// TwinCAT 3 PLC project PLC1
// ProgramVersion: 3.1.4022.4
// libraries:
//   Tc2_EtherCAT, * (Beckhoff Automation GmbH)
//   Tc2_IoFunctions, * (Beckhoff Automation GmbH)
//   Tc2_MC2, * (Beckhoff Automation GmbH)
//   Tc2_MC2_Camming, * (Beckhoff Automation GmbH)
//   Tc2_MDP, * (Beckhoff Automation GmbH)
//   Tc2_Standard, * (Beckhoff Automation GmbH)
//   Tc2_System, * (Beckhoff Automation GmbH)
//   Tc2_TcpIp, * (Beckhoff Automation GmbH)
//   Tc2_Utilities, * (Beckhoff Automation GmbH)
//   Tc3_Module, * (Beckhoff Automation GmbH)
//   VisuDialogs, * (System)
//   VisuSymbols,3.5.10.0,System
// project tree:
//   Add-On-Instructions/ AOI_AxisAdmin.TcPOU, AOI_Bin.TcPOU, AOI_CountersAdmin.TcPOU, AOI_CylinderAdmin.TcPOU, AOI_DeltaScaraRobot.TcPOU, AOI_HeatBase.TcPOU, AOI_MS300Admin.TcPOU, AOI_SensorAdmin.TcPOU, AOI_DI.TcPOU, AOI_DO.TcPOU, AOI_Heat.TcPOU, AOI_Timer.TcPOU, AOI_VacuumAdmin.TcPOU, BLINK.TcPOU, ethercatinfo_read.TcPOU, PackMlv3_StateModel.TcPOU, SequenceTransfer.TcPOU, systeminfo_MDP_read.TcPOU
//   Data-Types/User-Defined/ Condition.TcDUT, Seq_Status.TcDUT, SocketConnect.TcDUT, UDT_BinBelt.TcDUT, UDT_BoxList.TcDUT, UDT_Hmi_AxisView.TcDUT, UDT_Hmi_OEE.TcDUT, UDT_Recipe.TcDUT, UDT_MS300Output.TcDUT, UDT_MS300Input.TcDUT, UDT_DirectMotor.TcDUT, UDT_EL3312.TcDUT, UDT_EVENT.TcDUT, UDT_AxisAdmin.TcDUT, UDT_AxisInput.TcDUT, UDT_AxisOutput.TcDUT, UDT_Box.TcDUT, UDT_CM_Condition.TcDUT, UDT_CylinderAdmin.TcDUT, UDT_CylinderInput.TcDUT, UDT_CylinderOutput.TcDUT, UDT_EM_Status.TcDUT, UDT_EM_Cmd.TcDUT, UDT_Counters.TcDUT, UDT_Hmi_Input.TcDUT, UDT_Hmi_Output.TcDUT, UDT_MS300Admin.TcDUT, UDT_MS300_REF.TcDUT, UDT_Bin.TcDUT, UDT_BinList.TcDUT, UDT_Scara.TcDUT, UDT_Scara_DI.TcDUT, UDT_Scara_DO.TcDUT, UDT_SensorAdmin.TcDUT, UDT_SensorInput.TcDUT, UDT_SensorOutput.TcDUT, UDT_UnitAdmin.TcDUT, UDT_Unit_Cmd.TcDUT, UDT_Unit_Status.TcDUT, UDT_VacuumAdmin.TcDUT, UDT_VacuumInput.TcDUT, UDT_VacuumOutput.TcDUT
//   / CommunicationTask.TcTTO, GlobalTextList.TcGTLO, IOTask.TcTTO, MotionTask.TcTTO, PlcTask1.TcTTO, 视图管理器.TcVMO (not stored)
//   POUs/Debug/ DebugPro.TcPOU
//   POUs/EtherCat/ EtherCatStates.TcPOU
//   POUs/GVLs/ ControllerTags.TcGVL
//   POUs/IO/ IO_Mapping.TcPOU
//   POUs/MG/ MotionControl.TcPOU
//   POUs/PackMaL_UN01/ EM01_Master.TcPOU, EM02_Follower1.TcPOU, EM03_Follower2.TcPOU, EM04_Follower3.TcPOU, EM05_Counters.TcPOU, EM06_Follower4_5.TcPOU, EM07_Belt6.TcPOU, EM08_Belt7.TcPOU, UN01.TcPOU
//   POUs/POUCheck/ CheckBounds.TcPOU, CheckDivDInt.TcPOU, CheckDivLInt.TcPOU, CheckDivLReal.TcPOU, CheckDivReal.TcPOU, CheckLRangeSigned.TcPOU, CheckLRangeUnsigned.TcPOU, CheckPointer.TcPOU, CheckRangeSigned.TcPOU, CheckRangeUnsigned.TcPOU
//   POUs/Socket/ Socket.TcPOU
//   VISUs/ EM.TcVIS, Vis_MAIN.TcVIS, Vis_RealAxis.TcVIS, Vis_VirtualAxis.TcVIS
//   VISUs/Part/ Visualization_Cnt.TcVIS, Vis_Axis.TcVIS, Vis_PackMlv3.TcVIS
// real-time tasks:
//   TASK PlcTask1: cycle T#10ms, priority 14, ADS port 350
//   TASK CommunicationTask: cycle T#10ms, priority 16, ADS port 351
//   TASK MotionTask: cycle T#2ms, priority 6, ADS port 352
//   TASK IOTask: cycle T#2ms, priority 8, ADS port 353
//   TASK DataTask: cycle T#50000us, priority 18, ADS port 354
//   TASK Standard: cycle T#10ms, priority 20, ADS port 355
// motion (NC):
//   TASK NC-Task 1 SAF: cycle T#2ms, priority 4, ADS port 501
//   TASK NC-Task 1 SVB: cycle T#10ms, priority 12, ADS port 511
//   AXIS V_Master (id 100)
//     General: UnitFlags=#x00000004
//     Velo: Maximum=1000
//     OtherSettings: AllowMotionCmdToSlave=true
//     encoder EncType=1
//       EncPara: ModuloFactor=200
//     drive DrvType=5
//       Analog: VeloReferenz=1000, ScaleFactorActTorque=0.1
//       TimeComp: TaskDelayCycles=1
//     controller CtrType=1
//       CtrPara: PriorControlFactor=1
//         Observer: BandWidth=20
//   AXIS Belt 4 (id 2)
//     Velo: RefSearch=35
//     OtherSettings: AllowMotionCmdToSlave=true
//     encoder EncType=19
//       EncPara: ScaleFactorNumerator=40, ScaleFactorDenominator=1280000, ModuloFactor=3300, MaxCount=#xffffffff
//     drive DrvType=16
//       DrvPara: MaxCount=#xffffffff, DriveControlDWord=#x00020100
//         Analog: ScaleFactorActTorque=0.1
//         TimeComp: TaskDelayCycles=1
//     controller CtrType=1
//       CtrPara: PriorControlFactor=1
//         Observer: BandWidth=20
//   AXIS Belt 5 (id 3)
//     Velo: RefSearch=35
//     OtherSettings: AllowMotionCmdToSlave=true
//     encoder EncType=19
//       EncPara: ScaleFactorNumerator=40, ScaleFactorDenominator=1280000, ModuloFactor=3300, MaxCount=#xffffffff
//     drive DrvType=16
//       DrvPara: MaxCount=#xffffffff, DriveControlDWord=#x00020100
//         Analog: ScaleFactorActTorque=0.1
//         TimeComp: TaskDelayCycles=1
//     controller CtrType=1
//       CtrPara: PriorControlFactor=1
//         Observer: BandWidth=20
//   AXIS Belt 6 (id 4)
//     OtherSettings: AllowMotionCmdToSlave=true
//     encoder EncType=19
//       EncPara: ScaleFactorNumerator=18.0975, ScaleFactorDenominator=1280000, Inverse=true, MaxCount=#xffffffff
//     drive DrvType=16
//       DrvPara: Inverse=true, MaxCount=#xffffffff, DriveControlDWord=#x00020100
//         Analog: ScaleFactorActTorque=0.1
//         TimeComp: TaskDelayCycles=1
//     controller CtrType=1
//       CtrPara: PriorControlFactor=1
//         Observer: BandWidth=20
//   AXIS Counter 31 (id 5)
//     General: UnitName=Degree
//     Dynamic: AccelerationMaximum=450000, DecelerationMaximum=450000
//     Velo: Maximum=20000
//     OtherSettings: AllowMotionCmdToSlave=true
//     encoder EncType=19
//       EncPara: ScaleFactorNumerator=360, ScaleFactorDenominator=1280000, MaxCount=#xffffffff
//     drive DrvType=16
//       DrvPara: MaxCount=#xffffffff, DriveControlDWord=#x00020100
//         Analog: VeloReferenz=22000, ScaleFactorActTorque=0.1
//         TimeComp: TaskDelayCycles=1
//     controller CtrType=1
//       CtrPara: PriorControlFactor=1
//         Observer: BandWidth=20
//   AXIS Counter 32 (id 6)
//     Dynamic: AccelerationMaximum=450000, DecelerationMaximum=450000
//     Velo: Maximum=20000
//     OtherSettings: AllowMotionCmdToSlave=true
//     encoder EncType=19
//       EncPara: ScaleFactorNumerator=360, ScaleFactorDenominator=1280000, MaxCount=#xffffffff
//     drive DrvType=16
//       DrvPara: MaxCount=#xffffffff, DriveControlDWord=#x00020100
//         Analog: VeloReferenz=22000, ScaleFactorActTorque=0.1
//         TimeComp: TaskDelayCycles=1
//     controller CtrType=1
//       CtrPara: PriorControlFactor=1
//         Observer: BandWidth=20
//   AXIS Counter 33 (id 7)
//     Dynamic: AccelerationMaximum=450000, DecelerationMaximum=450000
//     Velo: Maximum=20000
//     OtherSettings: AllowMotionCmdToSlave=true
//     encoder EncType=19
//       EncPara: ScaleFactorNumerator=360, ScaleFactorDenominator=1280000, MaxCount=#xffffffff
//     drive DrvType=16
//       DrvPara: MaxCount=#xffffffff, DriveControlDWord=#x00020100
//         Analog: VeloReferenz=22000, ScaleFactorActTorque=0.1
//         TimeComp: TaskDelayCycles=1
//     controller CtrType=1
//       CtrPara: PriorControlFactor=1
//         Observer: BandWidth=20
//   AXIS Counter 34 (id 8)
//     Dynamic: AccelerationMaximum=450000, DecelerationMaximum=450000
//     Velo: Maximum=20000
//     OtherSettings: AllowMotionCmdToSlave=true
//     encoder EncType=19
//       EncPara: ScaleFactorNumerator=360, ScaleFactorDenominator=1280000, MaxCount=#xffffffff
//     drive DrvType=16
//       DrvPara: MaxCount=#xffffffff, DriveControlDWord=#x00020100
//         Analog: VeloReferenz=22000, ScaleFactorActTorque=0.1
//         TimeComp: TaskDelayCycles=1
//     controller CtrType=1
//       CtrPara: PriorControlFactor=1
//         Observer: BandWidth=20
//   AXIS Counter 35 (id 9)
//     Dynamic: AccelerationMaximum=450000, DecelerationMaximum=450000
//     Velo: Maximum=20000
//     OtherSettings: AllowMotionCmdToSlave=true
//     encoder EncType=19
//       EncPara: ScaleFactorNumerator=360, ScaleFactorDenominator=1280000, MaxCount=#xffffffff
//     drive DrvType=16
//       DrvPara: MaxCount=#xffffffff, DriveControlDWord=#x00020100
//         Analog: VeloReferenz=22000, ScaleFactorActTorque=0.1
//         TimeComp: TaskDelayCycles=1
//     controller CtrType=1
//       CtrPara: PriorControlFactor=1
//         Observer: BandWidth=20
//   AXIS Counter 36 (id 10)
//     Dynamic: AccelerationMaximum=450000, DecelerationMaximum=450000
//     Velo: Maximum=20000
//     OtherSettings: AllowMotionCmdToSlave=true
//     encoder EncType=19
//       EncPara: ScaleFactorNumerator=360, ScaleFactorDenominator=1280000, MaxCount=#xffffffff
//     drive DrvType=16
//       DrvPara: MaxCount=#xffffffff, DriveControlDWord=#x00020100
//         Analog: VeloReferenz=22000, ScaleFactorActTorque=0.1
//         TimeComp: TaskDelayCycles=1
//     controller CtrType=1
//       CtrPara: PriorControlFactor=1
//         Observer: BandWidth=20
//   AXIS Counter 37 (id 11)
//     Dynamic: AccelerationMaximum=450000, DecelerationMaximum=450000
//     Velo: Maximum=20000
//     OtherSettings: AllowMotionCmdToSlave=true
//     encoder EncType=19
//       EncPara: ScaleFactorNumerator=360, ScaleFactorDenominator=1280000, MaxCount=#xffffffff
//     drive DrvType=16
//       DrvPara: MaxCount=#xffffffff, DriveControlDWord=#x00020100
//         Analog: VeloReferenz=22000, ScaleFactorActTorque=0.1
//         TimeComp: TaskDelayCycles=1
//     controller CtrType=1
//       CtrPara: PriorControlFactor=1
//         Observer: BandWidth=20
//   AXIS Counter 38 (id 12)
//     Dynamic: AccelerationMaximum=450000, DecelerationMaximum=450000
//     Velo: Maximum=20000
//     OtherSettings: AllowMotionCmdToSlave=true
//     encoder EncType=19
//       EncPara: ScaleFactorNumerator=360, ScaleFactorDenominator=1280000, MaxCount=#xffffffff
//     drive DrvType=16
//       DrvPara: MaxCount=#xffffffff, DriveControlDWord=#x00020100
//         Analog: VeloReferenz=22000, ScaleFactorActTorque=0.1
//         TimeComp: TaskDelayCycles=1
//     controller CtrType=1
//       CtrPara: PriorControlFactor=1
//         Observer: BandWidth=20
//   AXIS Counter 39 (id 13)
//     Dynamic: AccelerationMaximum=450000, DecelerationMaximum=450000
//     Velo: Maximum=20000
//     OtherSettings: AllowMotionCmdToSlave=true
//     encoder EncType=19
//       EncPara: ScaleFactorNumerator=360, ScaleFactorDenominator=1280000, MaxCount=#xffffffff
//     drive DrvType=16
//       DrvPara: MaxCount=#xffffffff, DriveControlDWord=#x00020100
//         Analog: VeloReferenz=22000, ScaleFactorActTorque=0.1
//         TimeComp: TaskDelayCycles=1
//     controller CtrType=1
//       CtrPara: PriorControlFactor=1
//         Observer: BandWidth=20
//   AXIS Counter 40 (id 14)
//     Dynamic: AccelerationMaximum=450000, DecelerationMaximum=450000
//     Velo: Maximum=20000
//     OtherSettings: AllowMotionCmdToSlave=true
//     encoder EncType=19
//       EncPara: ScaleFactorNumerator=360, ScaleFactorDenominator=1280000, MaxCount=#xffffffff
//     drive DrvType=16
//       DrvPara: MaxCount=#xffffffff, DriveControlDWord=#x00020100
//         Analog: VeloReferenz=22000, ScaleFactorActTorque=0.1
//         TimeComp: TaskDelayCycles=1
//     controller CtrType=1
//       CtrPara: PriorControlFactor=1
//         Observer: BandWidth=20
//   AXIS Belt 3 (id 15)
//     Velo: RefSearch=40
//     OtherSettings: AllowMotionCmdToSlave=true
//     encoder EncType=19
//       EncPara: ScaleFactorNumerator=40, ScaleFactorDenominator=1280000, MaxCount=#xffffffff
//     drive DrvType=16
//       DrvPara: MaxCount=#xffffffff, DriveControlDWord=#x00020100
//         Analog: ScaleFactorActTorque=0.1
//         TimeComp: TaskDelayCycles=1
//     controller CtrType=1
//       CtrPara: PriorControlFactor=1
//         Observer: BandWidth=20
//   AXIS Counter 21 (id 16)
//     Dynamic: AccelerationMaximum=450000, DecelerationMaximum=450000
//     Velo: Maximum=20000
//     OtherSettings: AllowMotionCmdToSlave=true
//     encoder EncType=19
//       EncPara: ScaleFactorNumerator=360, ScaleFactorDenominator=1280000, MaxCount=#xffffffff
//     drive DrvType=16
//       DrvPara: MaxCount=#xffffffff, DriveControlDWord=#x00020100
//         Analog: VeloReferenz=22000, ScaleFactorActTorque=0.1
//         TimeComp: TaskDelayCycles=1
//     controller CtrType=1
//       CtrPara: PriorControlFactor=1
//         Observer: BandWidth=20
//   AXIS Counter 22 (id 17)
//     Dynamic: AccelerationMaximum=450000, DecelerationMaximum=450000
//     Velo: Maximum=20000
//     OtherSettings: AllowMotionCmdToSlave=true
//     encoder EncType=19
//       EncPara: ScaleFactorNumerator=360, ScaleFactorDenominator=1280000, MaxCount=#xffffffff
//     drive DrvType=16
//       DrvPara: MaxCount=#xffffffff, DriveControlDWord=#x00020100
//         Analog: VeloReferenz=22000, ScaleFactorActTorque=0.1
//         TimeComp: TaskDelayCycles=1
//     controller CtrType=1
//       CtrPara: PriorControlFactor=1
//         Observer: BandWidth=20
//   AXIS Counter 27 (id 22)
//     Dynamic: AccelerationMaximum=450000, DecelerationMaximum=450000
//     Velo: Maximum=20000
//     OtherSettings: AllowMotionCmdToSlave=true
//     encoder EncType=19
//       EncPara: ScaleFactorNumerator=360, ScaleFactorDenominator=1280000, MaxCount=#xffffffff
//     drive DrvType=16
//       DrvPara: MaxCount=#xffffffff, DriveControlDWord=#x00020100
//         Analog: VeloReferenz=22000, ScaleFactorActTorque=0.1
//         TimeComp: TaskDelayCycles=1
//     controller CtrType=1
//       CtrPara: PriorControlFactor=1
//         Observer: BandWidth=20
//   AXIS Counter 23 (id 18)
//     Dynamic: AccelerationMaximum=450000, DecelerationMaximum=450000
//     Velo: Maximum=20000
//     OtherSettings: AllowMotionCmdToSlave=true
//     encoder EncType=19
//       EncPara: ScaleFactorNumerator=360, ScaleFactorDenominator=1280000, MaxCount=#xffffffff
//     drive DrvType=16
//       DrvPara: MaxCount=#xffffffff, DriveControlDWord=#x00020100
//         Analog: VeloReferenz=22000, ScaleFactorActTorque=0.1
//         TimeComp: TaskDelayCycles=1
//     controller CtrType=1
//       CtrPara: PriorControlFactor=1
//         Observer: BandWidth=20
//   AXIS Counter 24 (id 19)
//     Dynamic: AccelerationMaximum=450000, DecelerationMaximum=450000
//     Velo: Maximum=20000
//     OtherSettings: AllowMotionCmdToSlave=true
//     encoder EncType=19
//       EncPara: ScaleFactorNumerator=360, ScaleFactorDenominator=1280000, MaxCount=#xffffffff
//     drive DrvType=16
//       DrvPara: MaxCount=#xffffffff, DriveControlDWord=#x00020100
//         Analog: VeloReferenz=22000, ScaleFactorActTorque=0.1
//         TimeComp: TaskDelayCycles=1
//     controller CtrType=1
//       CtrPara: PriorControlFactor=1
//         Observer: BandWidth=20
//   AXIS Counter 25 (id 20)
//     Dynamic: AccelerationMaximum=450000, DecelerationMaximum=450000
//     Velo: Maximum=20000
//     OtherSettings: AllowMotionCmdToSlave=true
//     encoder EncType=19
//       EncPara: ScaleFactorNumerator=360, ScaleFactorDenominator=1280000, MaxCount=#xffffffff
//     drive DrvType=16
//       DrvPara: MaxCount=#xffffffff, DriveControlDWord=#x00020100
//         Analog: VeloReferenz=22000, ScaleFactorActTorque=0.1
//         TimeComp: TaskDelayCycles=1
//     controller CtrType=1
//       CtrPara: PriorControlFactor=1
//         Observer: BandWidth=20
//   AXIS Counter 26 (id 21)
//     Dynamic: AccelerationMaximum=450000, DecelerationMaximum=450000
//     Velo: Maximum=20000
//     OtherSettings: AllowMotionCmdToSlave=true
//     encoder EncType=19
//       EncPara: ScaleFactorNumerator=360, ScaleFactorDenominator=1280000, MaxCount=#xffffffff
//     drive DrvType=16
//       DrvPara: MaxCount=#xffffffff, DriveControlDWord=#x00020100
//         Analog: VeloReferenz=22000, ScaleFactorActTorque=0.1
//         TimeComp: TaskDelayCycles=1
//     controller CtrType=1
//       CtrPara: PriorControlFactor=1
//         Observer: BandWidth=20
//   AXIS Counter 28 (id 23)
//     Dynamic: AccelerationMaximum=450000, DecelerationMaximum=450000
//     Velo: Maximum=20000
//     OtherSettings: AllowMotionCmdToSlave=true
//     encoder EncType=19
//       EncPara: ScaleFactorNumerator=360, ScaleFactorDenominator=1280000, MaxCount=#xffffffff
//     drive DrvType=16
//       DrvPara: MaxCount=#xffffffff, DriveControlDWord=#x00020100
//         Analog: VeloReferenz=22000, ScaleFactorActTorque=0.1
//         TimeComp: TaskDelayCycles=1
//     controller CtrType=1
//       CtrPara: PriorControlFactor=1
//         Observer: BandWidth=20
//   AXIS Counter 29 (id 24)
//     Dynamic: AccelerationMaximum=450000, DecelerationMaximum=450000
//     Velo: Maximum=20000
//     OtherSettings: AllowMotionCmdToSlave=true
//     encoder EncType=19
//       EncPara: ScaleFactorNumerator=360, ScaleFactorDenominator=1280000, MaxCount=#xffffffff
//     drive DrvType=16
//       DrvPara: MaxCount=#xffffffff, DriveControlDWord=#x00020100
//         Analog: VeloReferenz=22000, ScaleFactorActTorque=0.1
//         TimeComp: TaskDelayCycles=1
//     controller CtrType=1
//       CtrPara: PriorControlFactor=1
//         Observer: BandWidth=20
//   AXIS Counter 30 (id 25)
//     Dynamic: AccelerationMaximum=450000, DecelerationMaximum=450000
//     Velo: Maximum=20000
//     OtherSettings: AllowMotionCmdToSlave=true
//     encoder EncType=19
//       EncPara: ScaleFactorNumerator=360, ScaleFactorDenominator=1280000, MaxCount=#xffffffff
//     drive DrvType=16
//       DrvPara: MaxCount=#xffffffff, DriveControlDWord=#x00020100
//         Analog: VeloReferenz=22000, ScaleFactorActTorque=0.1
//         TimeComp: TaskDelayCycles=1
//     controller CtrType=1
//       CtrPara: PriorControlFactor=1
//         Observer: BandWidth=20
//   AXIS Belt 2 (id 26)
//     Velo: RefSearch=40
//     OtherSettings: AllowMotionCmdToSlave=true
//     encoder EncType=19
//       EncPara: ScaleFactorNumerator=40, ScaleFactorDenominator=1280000, MaxCount=#xffffffff
//     drive DrvType=16
//       DrvPara: MaxCount=#xffffffff, DriveControlDWord=#x00020100
//         Analog: ScaleFactorActTorque=0.1
//         TimeComp: TaskDelayCycles=1
//     controller CtrType=1
//       CtrPara: PriorControlFactor=1
//         Observer: BandWidth=20
//   AXIS Counter 11 (id 27)
//     Dynamic: AccelerationMaximum=450000, DecelerationMaximum=450000
//     Velo: Maximum=20000
//     OtherSettings: AllowMotionCmdToSlave=true
//     encoder EncType=19
//       EncPara: ScaleFactorNumerator=360, ScaleFactorDenominator=1280000, MaxCount=#xffffffff
//     drive DrvType=16
//       DrvPara: MaxCount=#xffffffff, DriveControlDWord=#x00020100
//         Analog: VeloReferenz=22000, ScaleFactorActTorque=0.1
//         TimeComp: TaskDelayCycles=1
//     controller CtrType=1
//       CtrPara: PriorControlFactor=1
//         Observer: BandWidth=20
//   AXIS Counter 12 (id 28)
//     Dynamic: AccelerationMaximum=450000, DecelerationMaximum=450000
//     Velo: Maximum=20000
//     OtherSettings: AllowMotionCmdToSlave=true
//     encoder EncType=19
//       EncPara: ScaleFactorNumerator=360, ScaleFactorDenominator=1280000, MaxCount=#xffffffff
//     drive DrvType=16
//       DrvPara: MaxCount=#xffffffff, DriveControlDWord=#x00020100
//         Analog: VeloReferenz=22000, ScaleFactorActTorque=0.1
//         TimeComp: TaskDelayCycles=1
//     controller CtrType=1
//       CtrPara: PriorControlFactor=1
//         Observer: BandWidth=20
//   AXIS Counter 13 (id 29)
//     Dynamic: AccelerationMaximum=450000, DecelerationMaximum=450000
//     Velo: Maximum=20000
//     OtherSettings: AllowMotionCmdToSlave=true
//     encoder EncType=19
//       EncPara: ScaleFactorNumerator=360, ScaleFactorDenominator=1280000, MaxCount=#xffffffff
//     drive DrvType=16
//       DrvPara: MaxCount=#xffffffff, DriveControlDWord=#x00020100
//         Analog: VeloReferenz=22000, ScaleFactorActTorque=0.1
//         TimeComp: TaskDelayCycles=1
//     controller CtrType=1
//       CtrPara: PriorControlFactor=1
//         Observer: BandWidth=20
//   AXIS Counter 14 (id 30)
//     Dynamic: AccelerationMaximum=450000, DecelerationMaximum=450000
//     Velo: Maximum=20000
//     OtherSettings: AllowMotionCmdToSlave=true
//     encoder EncType=19
//       EncPara: ScaleFactorNumerator=360, ScaleFactorDenominator=1280000, MaxCount=#xffffffff
//     drive DrvType=16
//       DrvPara: MaxCount=#xffffffff, DriveControlDWord=#x00020100
//         Analog: VeloReferenz=22000, ScaleFactorActTorque=0.1
//         TimeComp: TaskDelayCycles=1
//     controller CtrType=1
//       CtrPara: PriorControlFactor=1
//         Observer: BandWidth=20
//   AXIS Counter 15 (id 31)
//     Dynamic: AccelerationMaximum=450000, DecelerationMaximum=450000
//     Velo: Maximum=20000
//     OtherSettings: AllowMotionCmdToSlave=true
//     encoder EncType=19
//       EncPara: ScaleFactorNumerator=360, ScaleFactorDenominator=1280000, MaxCount=#xffffffff
//     drive DrvType=16
//       DrvPara: MaxCount=#xffffffff, DriveControlDWord=#x00020100
//         Analog: VeloReferenz=22000, ScaleFactorActTorque=0.1
//         TimeComp: TaskDelayCycles=1
//     controller CtrType=1
//       CtrPara: PriorControlFactor=1
//         Observer: BandWidth=20
//   AXIS Counter 16 (id 32)
//     Dynamic: AccelerationMaximum=450000, DecelerationMaximum=450000
//     Velo: Maximum=20000
//     OtherSettings: AllowMotionCmdToSlave=true
//     encoder EncType=19
//       EncPara: ScaleFactorNumerator=360, ScaleFactorDenominator=1280000, MaxCount=#xffffffff
//     drive DrvType=16
//       DrvPara: MaxCount=#xffffffff, DriveControlDWord=#x00020100
//         Analog: VeloReferenz=22000, ScaleFactorActTorque=0.1
//         TimeComp: TaskDelayCycles=1
//     controller CtrType=1
//       CtrPara: PriorControlFactor=1
//         Observer: BandWidth=20
//   AXIS Counter 17 (id 33)
//     Dynamic: AccelerationMaximum=450000, DecelerationMaximum=450000
//     Velo: Maximum=20000
//     OtherSettings: AllowMotionCmdToSlave=true
//     encoder EncType=19
//       EncPara: ScaleFactorNumerator=360, ScaleFactorDenominator=1280000, MaxCount=#xffffffff
//     drive DrvType=16
//       DrvPara: MaxCount=#xffffffff, DriveControlDWord=#x00020100
//         Analog: VeloReferenz=22000, ScaleFactorActTorque=0.1
//         TimeComp: TaskDelayCycles=1
//     controller CtrType=1
//       CtrPara: PriorControlFactor=1
//         Observer: BandWidth=20
//   AXIS Counter 18 (id 34)
//     Dynamic: AccelerationMaximum=450000, DecelerationMaximum=450000
//     Velo: Maximum=20000
//     OtherSettings: AllowMotionCmdToSlave=true
//     encoder EncType=19
//       EncPara: ScaleFactorNumerator=360, ScaleFactorDenominator=1280000, MaxCount=#xffffffff
//     drive DrvType=16
//       DrvPara: MaxCount=#xffffffff, DriveControlDWord=#x00020100
//         Analog: VeloReferenz=22000, ScaleFactorActTorque=0.1
//         TimeComp: TaskDelayCycles=1
//     controller CtrType=1
//       CtrPara: PriorControlFactor=1
//         Observer: BandWidth=20
//   AXIS Counter 19 (id 35)
//     Dynamic: AccelerationMaximum=450000, DecelerationMaximum=450000
//     Velo: Maximum=20000
//     OtherSettings: AllowMotionCmdToSlave=true
//     encoder EncType=19
//       EncPara: ScaleFactorNumerator=360, ScaleFactorDenominator=1280000, MaxCount=#xffffffff
//     drive DrvType=16
//       DrvPara: MaxCount=#xffffffff, DriveControlDWord=#x00020100
//         Analog: VeloReferenz=22000, ScaleFactorActTorque=0.1
//         TimeComp: TaskDelayCycles=1
//     controller CtrType=1
//       CtrPara: PriorControlFactor=1
//         Observer: BandWidth=20
//   AXIS Counter 20 (id 36)
//     Dynamic: AccelerationMaximum=450000, DecelerationMaximum=450000
//     Velo: Maximum=20000
//     OtherSettings: AllowMotionCmdToSlave=true
//     encoder EncType=19
//       EncPara: ScaleFactorNumerator=360, ScaleFactorDenominator=1280000, MaxCount=#xffffffff
//     drive DrvType=16
//       DrvPara: MaxCount=#xffffffff, DriveControlDWord=#x00020100
//         Analog: VeloReferenz=22000, ScaleFactorActTorque=0.1
//         TimeComp: TaskDelayCycles=1
//     controller CtrType=1
//       CtrPara: PriorControlFactor=1
//         Observer: BandWidth=20
//   AXIS Belt 1 (id 37)
//     Velo: RefSearch=40
//     OtherSettings: AllowMotionCmdToSlave=true
//     encoder EncType=19
//       EncPara: ScaleFactorNumerator=40, ScaleFactorDenominator=1280000, MaxCount=#xffffffff
//     drive DrvType=16
//       DrvPara: MaxCount=#xffffffff, DriveControlDWord=#x00020100
//         Analog: ScaleFactorActTorque=0.1
//         TimeComp: TaskDelayCycles=1
//     controller CtrType=1
//       CtrPara: PriorControlFactor=1
//         Observer: BandWidth=20
//   AXIS Counter 1 (id 38)
//     General: UnitName=Degree
//     Dynamic: AccelerationMaximum=450000, DecelerationMaximum=450000
//     Velo: Maximum=20000
//     OtherSettings: AllowMotionCmdToSlave=true
//     encoder EncType=19
//       EncPara: ScaleFactorNumerator=360, ScaleFactorDenominator=1280000, MaxCount=#xffffffff
//     drive DrvType=16
//       DrvPara: MaxCount=#xffffffff, DriveControlDWord=#x00020100
//         Analog: VeloReferenz=22000, ScaleFactorActTorque=0.1
//         TimeComp: TaskDelayCycles=1
//     controller CtrType=1
//       CtrPara: PriorControlFactor=1
//         Observer: BandWidth=20
//   AXIS Counter 2 (id 39)
//     General: UnitName=Degree
//     Dynamic: AccelerationMaximum=450000, DecelerationMaximum=450000
//     Velo: Maximum=20000
//     OtherSettings: AllowMotionCmdToSlave=true
//     encoder EncType=19
//       EncPara: ScaleFactorNumerator=360, ScaleFactorDenominator=1280000, MaxCount=#xffffffff
//     drive DrvType=16
//       DrvPara: MaxCount=#xffffffff, DriveControlDWord=#x00020100
//         Analog: VeloReferenz=22000, ScaleFactorActTorque=0.1
//         TimeComp: TaskDelayCycles=1
//     controller CtrType=1
//       CtrPara: PriorControlFactor=1
//         Observer: BandWidth=20
//   AXIS Counter 3 (id 40)
//     General: UnitName=Degree
//     Dynamic: AccelerationMaximum=450000, DecelerationMaximum=450000
//     Velo: Maximum=20000
//     OtherSettings: AllowMotionCmdToSlave=true
//     encoder EncType=19
//       EncPara: ScaleFactorNumerator=360, ScaleFactorDenominator=1280000, MaxCount=#xffffffff
//     drive DrvType=16
//       DrvPara: MaxCount=#xffffffff, DriveControlDWord=#x00020100
//         Analog: VeloReferenz=22000, ScaleFactorActTorque=0.1
//         TimeComp: TaskDelayCycles=1
//     controller CtrType=1
//       CtrPara: PriorControlFactor=1
//         Observer: BandWidth=20
//   AXIS Counter 4 (id 41)
//     Dynamic: AccelerationMaximum=450000, DecelerationMaximum=450000
//     Velo: Maximum=20000
//     OtherSettings: AllowMotionCmdToSlave=true
//     encoder EncType=19
//       EncPara: ScaleFactorNumerator=360, ScaleFactorDenominator=1280000, MaxCount=#xffffffff
//     drive DrvType=16
//       DrvPara: MaxCount=#xffffffff, DriveControlDWord=#x00020100
//         Analog: VeloReferenz=22000, ScaleFactorActTorque=0.1
//         TimeComp: TaskDelayCycles=1
//     controller CtrType=1
//       CtrPara: PriorControlFactor=1
//         Observer: BandWidth=20
//   AXIS Counter 5 (id 42)
//     Dynamic: AccelerationMaximum=450000, DecelerationMaximum=450000
//     Velo: Maximum=20000
//     OtherSettings: AllowMotionCmdToSlave=true
//     encoder EncType=19
//       EncPara: ScaleFactorNumerator=360, ScaleFactorDenominator=1280000, MaxCount=#xffffffff
//     drive DrvType=16
//       DrvPara: MaxCount=#xffffffff, DriveControlDWord=#x00020100
//         Analog: VeloReferenz=22000, ScaleFactorActTorque=0.1
//         TimeComp: TaskDelayCycles=1
//     controller CtrType=1
//       CtrPara: PriorControlFactor=1
//         Observer: BandWidth=20
//   AXIS Counter 6 (id 43)
//     Dynamic: AccelerationMaximum=450000, DecelerationMaximum=450000
//     Velo: Maximum=20000
//     OtherSettings: AllowMotionCmdToSlave=true
//     encoder EncType=19
//       EncPara: ScaleFactorNumerator=360, ScaleFactorDenominator=1280000, MaxCount=#xffffffff
//     drive DrvType=16
//       DrvPara: MaxCount=#xffffffff, DriveControlDWord=#x00020100
//         Analog: VeloReferenz=22000, ScaleFactorActTorque=0.1
//         TimeComp: TaskDelayCycles=1
//     controller CtrType=1
//       CtrPara: PriorControlFactor=1
//         Observer: BandWidth=20
//   AXIS Counter 7 (id 44)
//     Dynamic: AccelerationMaximum=450000, DecelerationMaximum=450000
//     Velo: Maximum=20000
//     OtherSettings: AllowMotionCmdToSlave=true
//     encoder EncType=19
//       EncPara: ScaleFactorNumerator=360, ScaleFactorDenominator=1280000, MaxCount=#xffffffff
//     drive DrvType=16
//       DrvPara: MaxCount=#xffffffff, DriveControlDWord=#x00020100
//         Analog: VeloReferenz=22000, ScaleFactorActTorque=0.1
//         TimeComp: TaskDelayCycles=1
//     controller CtrType=1
//       CtrPara: PriorControlFactor=1
//         Observer: BandWidth=20
//   AXIS Counter 8 (id 45)
//     Dynamic: AccelerationMaximum=450000, DecelerationMaximum=450000
//     Velo: Maximum=20000
//     OtherSettings: AllowMotionCmdToSlave=true
//     encoder EncType=19
//       EncPara: ScaleFactorNumerator=360, ScaleFactorDenominator=1280000, MaxCount=#xffffffff
//     drive DrvType=16
//       DrvPara: MaxCount=#xffffffff, DriveControlDWord=#x00020100
//         Analog: VeloReferenz=22000, ScaleFactorActTorque=0.1
//         TimeComp: TaskDelayCycles=1
//     controller CtrType=1
//       CtrPara: PriorControlFactor=1
//         Observer: BandWidth=20
//   AXIS Counter 9 (id 46)
//     Dynamic: AccelerationMaximum=450000, DecelerationMaximum=450000
//     Velo: Maximum=20000
//     OtherSettings: AllowMotionCmdToSlave=true
//     encoder EncType=19
//       EncPara: ScaleFactorNumerator=360, ScaleFactorDenominator=1280000, MaxCount=#xffffffff
//     drive DrvType=16
//       DrvPara: MaxCount=#xffffffff, DriveControlDWord=#x00020100
//         Analog: VeloReferenz=22000, ScaleFactorActTorque=0.1
//         TimeComp: TaskDelayCycles=1
//     controller CtrType=1
//       CtrPara: PriorControlFactor=1
//         Observer: BandWidth=20
//   AXIS Counter 10 (id 47)
//     Dynamic: AccelerationMaximum=450000, DecelerationMaximum=450000
//     Velo: Maximum=20000
//     OtherSettings: AllowMotionCmdToSlave=true
//     encoder EncType=19
//       EncPara: ScaleFactorNumerator=360, ScaleFactorDenominator=1280000, MaxCount=#xffffffff
//     drive DrvType=16
//       DrvPara: MaxCount=#xffffffff, DriveControlDWord=#x00020100
//         Analog: VeloReferenz=22000, ScaleFactorActTorque=0.1
//         TimeComp: TaskDelayCycles=1
//     controller CtrType=1
//       CtrPara: PriorControlFactor=1
//         Observer: BandWidth=20
//   AXIS eAxis1 (id 101)
//     OtherSettings: AllowMotionCmdToSlave=true
//     encoder EncType=4
//       EncPara: ScaleFactorNumerator=157, ScaleFactorDenominator=1600, MaxCount=#x0000ffff
//         Inc: RefSoftSyncMask=#x0000ffff
//     drive DrvType=5
//       Analog: ScaleFactorActTorque=0.1
//       TimeComp: TaskDelayCycles=1
//     controller CtrType=1
//       CtrPara: PriorControlFactor=1
//         Observer: BandWidth=20
//   AXIS V_Master2 (id 102)
//     OtherSettings: AllowMotionCmdToSlave=true
//     encoder EncType=1
//     drive DrvType=5
//       Analog: ScaleFactorActTorque=0.1
//       TimeComp: TaskDelayCycles=1
//     controller CtrType=1
//       CtrPara: PriorControlFactor=1
//         Observer: BandWidth=20
//   AXIS Belt7 (id 48)
//     OtherSettings: AllowMotionCmdToSlave=true
//     encoder EncType=19
//       EncPara: ScaleFactorNumerator=16, ScaleFactorDenominator=1280000, Inverse=true, MaxCount=#xffffffff
//         Inc: RefSearchInverse=true
//     drive DrvType=16
//       DrvPara: Inverse=true, MaxCount=#xffffffff, DriveControlDWord=#x00020100
//         Analog: ScaleFactorActTorque=0.1
//         TimeComp: TaskDelayCycles=1
//     controller CtrType=1
//       CtrPara: PriorControlFactor=1
//         Observer: BandWidth=20
//   AXIS Puller (id 1)
//     OtherSettings: AllowMotionCmdToSlave=true
//     encoder EncType=19
//       EncPara: ScaleFactorNumerator=15.7, ScaleFactorDenominator=1280000, Inverse=true, MaxCount=#xffffffff
//     drive DrvType=16
//       DrvPara: Inverse=true, MaxCount=#xffffffff, DriveControlDWord=#x00020100
//         Analog: ScaleFactorActTorque=0.1
//         TimeComp: TaskDelayCycles=1
//     controller CtrType=1
//       CtrPara: PriorControlFactor=1
//         Observer: BandWidth=20
// I/O:
//   DEVICE Device 1 (EtherCAT), AmsNetId 5.74.170.4.2.1
//     Term 1 (EK1200) [EK1200-5000 EtherCAT Power supply (2A E-Bus)]
//       Term 2 (EL1008) [EL1008 8Ch. Dig. Input 24V, 3ms]
//       Term 3 (EL1008) [EL1008 8Ch. Dig. Input 24V, 3ms]
//       Term 4 (EL1008) [EL1008 8Ch. Dig. Input 24V, 3ms]
//       Term 5 (EL1008) [EL1008 8Ch. Dig. Input 24V, 3ms]
//       Term 6 (EL1008) [EL1008 8Ch. Dig. Input 24V, 3ms]
//       Term 7 (EL2008) [EL2008 8Ch. Dig. Output 24V, 0.5A]
//       Term 8 (EL2008) [EL2008 8Ch. Dig. Output 24V, 0.5A]
//       Term 9 (EL2008) [EL2008 8Ch. Dig. Output 24V, 0.5A]
//       Term 10 (EL2008) [EL2008 8Ch. Dig. Output 24V, 0.5A]
//       Term 11 (EL9410) [EL9410 E-Bus Power Supplier  (Diagnostics)]
//       Term 12 (EL3312) [EL3312 2Ch. Ana. Input Thermocouple (TC)]
//       Term 13 (EL3312) [EL3312 2Ch. Ana. Input Thermocouple (TC)]
//       Term 14 (EL3312) [EL3312 2Ch. Ana. Input Thermocouple (TC)]
//       Term 15 (EL3312) [EL3312 2Ch. Ana. Input Thermocouple (TC)]
//       Term 16 (EL5101) [EL5101 1Ch. Inc. Encoder 5V]
//       Term 17 (EK1122) [EK1122 2 port EtherCAT junction]
//         Drive PA14701 (ASDA-A2-E CoE Drive) [Delta ASDA-A2-E EtherCAT(CoE) Drive Rev4]
//         Drive PA14401 (ASDA-A2-E CoE Drive) [Delta ASDA-A2-E EtherCAT(CoE) Drive Rev4]
//         Drive PA14501 (ASDA-A2-E CoE Drive) [Delta ASDA-A2-E EtherCAT(CoE) Drive Rev4]
//         Drive PA14601 (ASDA-A2-E CoE Drive) [Delta ASDA-A2-E EtherCAT(CoE) Drive]
//         WPI_1(WPI_EtherCAt_32Bits) [WPI-32Bits]
//         WPI_2(WPI_EtherCAt_32Bits) [WPI-32Bits]
//         CPX_1 VI45001 (CPX-AP-I-EC-M12) [CPX-AP-I-EC-M12]
//           modules: Module 1 (CPX-AP-I-EC-M12), Module 2 (CPX-AP-I-8DI-M8-3P), Module 3 (CPX-AP-I-8DI-M8-3P), Module 4 (CPX-AP-I-8DI-M8-3P), Module 5 (CPX-AP-I-8DI-M8-3P), Module 6 (CPX-AP-I-8DI-M8-3P), Module 7 (CPX-AP-I-8DI-M8-3P), Module 8 (CPX-AP-I-8DI-M8-3P)
//       Term 22 (EK1110) [EK1110 EtherCAT extension]
//     Drive PA14901 (ASDA-A2-E CoE Drive) [Delta ASDA-A2-E EtherCAT(CoE) Drive Rev4]
//   DEVICE Device 4 (EtherCAT), AmsNetId 5.74.170.4.5.1
//     Drive PA13301 (ASDA-A2-E CoE Drive) [Delta ASDA-A2-E EtherCAT(CoE) Drive Rev4]
//     Drive PA13401 (ASDA-A2-E CoE Drive) [Delta ASDA-A2-E EtherCAT(CoE) Drive Rev4]
//     Drive PA13501 (ASDA-A2-E CoE Drive) [Delta ASDA-A2-E EtherCAT(CoE) Drive Rev4]
//     Drive PA13601 (ASDA-A2-E CoE Drive) [Delta ASDA-A2-E EtherCAT(CoE) Drive Rev4]
//     Drive PA13701 (ASDA-A2-E CoE Drive) [Delta ASDA-A2-E EtherCAT(CoE) Drive Rev4]
//     Term CIM36901 (EK1100) [EK1100 EtherCAT Coupler (2A E-Bus)]
//       Term 29 (EL1008) [EL1008 8Ch. Dig. Input 24V, 3ms]
//       Term 30 (EL1008) [EL1008 8Ch. Dig. Input 24V, 3ms]
//       Term 31 (EL1008) [EL1008 8Ch. Dig. Input 24V, 3ms]
//       Term 32 (EL1008) [EL1008 8Ch. Dig. Input 24V, 3ms]
//       Term 33 (EL1008) [EL1008 8Ch. Dig. Input 24V, 3ms]
//       Term 34 (EL1008) [EL1008 8Ch. Dig. Input 24V, 3ms]
//       Term 35 (EL1008) [EL1008 8Ch. Dig. Input 24V, 3ms]
//       Term 36 (EL1008) [EL1008 8Ch. Dig. Input 24V, 3ms]
//       Term 37 (EL2008) [EL2008 8Ch. Dig. Output 24V, 0.5A]
//       Term 38 (EL2008) [EL2008 8Ch. Dig. Output 24V, 0.5A]
//       Term 39 (EL2008) [EL2008 8Ch. Dig. Output 24V, 0.5A]
//       Term 40 (EL2008) [EL2008 8Ch. Dig. Output 24V, 0.5A]
//       Term 41 (EL2008) [EL2008 8Ch. Dig. Output 24V, 0.5A]
//       Term 42 (EL2008) [EL2008 8Ch. Dig. Output 24V, 0.5A]
//       Term 43 (EL2008) [EL2008 8Ch. Dig. Output 24V, 0.5A]
//       Term 108 (EL9011) [EL9011 End Terminal]
//     Drive PA13801 (ASDA-A2-E CoE Drive) [Delta ASDA-A2-E EtherCAT(CoE) Drive Rev4]
//     Drive PA13901 (ASDA-A2-E CoE Drive) [Delta ASDA-A2-E EtherCAT(CoE) Drive Rev4]
//     Drive PA14001 (ASDA-A2-E CoE Drive) [Delta ASDA-A2-E EtherCAT(CoE) Drive Rev4]
//     Drive PA14101 (ASDA-A2-E CoE Drive) [Delta ASDA-A2-E EtherCAT(CoE) Drive Rev4]
//     Drive PA14201 (ASDA-A2-E CoE Drive) [Delta ASDA-A2-E EtherCAT(CoE) Drive Rev4]
//     Drive PA14301 (ASDA-A2-E CoE Drive) [Delta ASDA-A2-E EtherCAT(CoE) Drive Rev4]
//     Drive PA12201 (ASDA-A2-E CoE Drive) [Delta ASDA-A2-E EtherCAT(CoE) Drive Rev4]
//     Drive PA12301 (ASDA-A2-E CoE Drive) [Delta ASDA-A2-E EtherCAT(CoE) Drive Rev4]
//     Drive PA12401 (ASDA-A2-E CoE Drive) [Delta ASDA-A2-E EtherCAT(CoE) Drive Rev4]
//     Drive PA12501 (ASDA-A2-E CoE Drive) [Delta ASDA-A2-E EtherCAT(CoE) Drive Rev4]
//     Drive PA12601 (ASDA-A2-E CoE Drive) [Delta ASDA-A2-E EtherCAT(CoE) Drive Rev4]
//     Term CIM35301 (EK1100) [EK1100 EtherCAT Coupler (2A E-Bus)]
//       Term 56 (EL1008) [EL1008 8Ch. Dig. Input 24V, 3ms]
//       Term 57 (EL1008) [EL1008 8Ch. Dig. Input 24V, 3ms]
//       Term 58 (EL1008) [EL1008 8Ch. Dig. Input 24V, 3ms]
//       Term 59 (EL1008) [EL1008 8Ch. Dig. Input 24V, 3ms]
//       Term 60 (EL1008) [EL1008 8Ch. Dig. Input 24V, 3ms]
//       Term 61 (EL1008) [EL1008 8Ch. Dig. Input 24V, 3ms]
//       Term 62 (EL1008) [EL1008 8Ch. Dig. Input 24V, 3ms]
//       Term 63 (EL1008) [EL1008 8Ch. Dig. Input 24V, 3ms]
//       Term 64 (EL2008) [EL2008 8Ch. Dig. Output 24V, 0.5A]
//       Term 65 (EL2008) [EL2008 8Ch. Dig. Output 24V, 0.5A]
//       Term 66 (EL2008) [EL2008 8Ch. Dig. Output 24V, 0.5A]
//       Term 67 (EL2008) [EL2008 8Ch. Dig. Output 24V, 0.5A]
//       Term 68 (EL2008) [EL2008 8Ch. Dig. Output 24V, 0.5A]
//       Term 69 (EL2008) [EL2008 8Ch. Dig. Output 24V, 0.5A]
//       Term 70 (EL2008) [EL2008 8Ch. Dig. Output 24V, 0.5A]
//       Term 109 (EL9011) [EL9011 End Terminal]
//     Drive PA12701 (ASDA-A2-E CoE Drive) [Delta ASDA-A2-E EtherCAT(CoE) Drive Rev4]
//     Drive PA12801 (ASDA-A2-E CoE Drive) [Delta ASDA-A2-E EtherCAT(CoE) Drive Rev4]
//     Drive PA12901 (ASDA-A2-E CoE Drive) [Delta ASDA-A2-E EtherCAT(CoE) Drive Rev4]
//     Drive PA13001 (ASDA-A2-E CoE Drive) [Delta ASDA-A2-E EtherCAT(CoE) Drive Rev4]
//     Drive PA13101 (ASDA-A2-E CoE Drive) [Delta ASDA-A2-E EtherCAT(CoE) Drive Rev4]
//     Drive PA13201 (ASDA-A2-E CoE Drive) [Delta ASDA-A2-E EtherCAT(CoE) Drive Rev4]
//     Drive PA11101 (ASDA-A2-E CoE Drive) [Delta ASDA-A2-E EtherCAT(CoE) Drive Rev4]
//     Drive PA11201 (ASDA-A2-E CoE Drive) [Delta ASDA-A2-E EtherCAT(CoE) Drive Rev4]
//     Drive PA11301 (ASDA-A2-E CoE Drive) [Delta ASDA-A2-E EtherCAT(CoE) Drive Rev4]
//     Drive PA11401 (ASDA-A2-E CoE Drive) [Delta ASDA-A2-E EtherCAT(CoE) Drive Rev4]
//     Drive PA11501 (ASDA-A2-E CoE Drive) [Delta ASDA-A2-E EtherCAT(CoE) Drive Rev4]
//     Term CIM33701 (EK1100) [EK1100 EtherCAT Coupler (2A E-Bus)]
//       Term 83 (EL1008) [EL1008 8Ch. Dig. Input 24V, 3ms]
//       Term 84 (EL1008) [EL1008 8Ch. Dig. Input 24V, 3ms]
//       Term 85 (EL1008) [EL1008 8Ch. Dig. Input 24V, 3ms]
//       Term 86 (EL1008) [EL1008 8Ch. Dig. Input 24V, 3ms]
//       Term 87 (EL1008) [EL1008 8Ch. Dig. Input 24V, 3ms]
//       Term 88 (EL1008) [EL1008 8Ch. Dig. Input 24V, 3ms]
//       Term 89 (EL1008) [EL1008 8Ch. Dig. Input 24V, 3ms]
//       Term 90 (EL1008) [EL1008 8Ch. Dig. Input 24V, 3ms]
//       Term 91 (EL2008) [EL2008 8Ch. Dig. Output 24V, 0.5A]
//       Term 92 (EL2008) [EL2008 8Ch. Dig. Output 24V, 0.5A]
//       Term 93 (EL2008) [EL2008 8Ch. Dig. Output 24V, 0.5A]
//       Term 94 (EL2008) [EL2008 8Ch. Dig. Output 24V, 0.5A]
//       Term 95 (EL2008) [EL2008 8Ch. Dig. Output 24V, 0.5A]
//       Term 96 (EL2008) [EL2008 8Ch. Dig. Output 24V, 0.5A]
//       Term 97 (EL2008) [EL2008 8Ch. Dig. Output 24V, 0.5A]
//       Term 110 (EL9011) [EL9011 End Terminal]
//     Drive PA11601 (ASDA-A2-E CoE Drive) [Delta ASDA-A2-E EtherCAT(CoE) Drive Rev4]
//     Drive PA11701 (ASDA-A2-E CoE Drive) [Delta ASDA-A2-E EtherCAT(CoE) Drive Rev4]
//     Drive PA11801 (ASDA-A2-E CoE Drive) [Delta ASDA-A2-E EtherCAT(CoE) Drive Rev4]
//     Drive PA11901 (ASDA-A2-E CoE Drive) [Delta ASDA-A2-E EtherCAT(CoE) Drive Rev4]
//     Drive PA12001 (ASDA-A2-E CoE Drive) [Delta ASDA-A2-E EtherCAT(CoE) Drive Rev4]
//     Drive PA12101 (ASDA-A2-E CoE Drive) [Delta ASDA-A2-E EtherCAT(CoE) Drive Rev4]
//     Drive PA10101 (ASDA-A2-E CoE Drive) [Delta ASDA-A2-E EtherCAT(CoE) Drive Rev4]
//     Drive PA10201 (ASDA-A2-E CoE Drive) [Delta ASDA-A2-E EtherCAT(CoE) Drive Rev4]
//     Drive PA10301 (ASDA-A2-E CoE Drive) [Delta ASDA-A2-E EtherCAT(CoE) Drive Rev4]
//     Drive PA10401 (ASDA-A2-E CoE Drive) [Delta ASDA-A2-E EtherCAT(CoE) Drive Rev4]
//     Drive PA10501 (ASDA-A2-E CoE Drive) [Delta ASDA-A2-E EtherCAT(CoE) Drive Rev4]
//     Term CIM32101 (EK1100) [EK1100 EtherCAT Coupler (2A E-Bus)]
//       Term 110 (EL1008) [EL1008 8Ch. Dig. Input 24V, 3ms]
//       Term 111 (EL1008) [EL1008 8Ch. Dig. Input 24V, 3ms]
//       Term 112 (EL1008) [EL1008 8Ch. Dig. Input 24V, 3ms]
//       Term 113 (EL1008) [EL1008 8Ch. Dig. Input 24V, 3ms]
//       Term 114 (EL1008) [EL1008 8Ch. Dig. Input 24V, 3ms]
//       Term 115 (EL1008) [EL1008 8Ch. Dig. Input 24V, 3ms]
//       Term 116 (EL1008) [EL1008 8Ch. Dig. Input 24V, 3ms]
//       Term 117 (EL1008) [EL1008 8Ch. Dig. Input 24V, 3ms]
//       Term 118 (EL2008) [EL2008 8Ch. Dig. Output 24V, 0.5A]
//       Term 119 (EL2008) [EL2008 8Ch. Dig. Output 24V, 0.5A]
//       Term 120 (EL2008) [EL2008 8Ch. Dig. Output 24V, 0.5A]
//       Term 121 (EL2008) [EL2008 8Ch. Dig. Output 24V, 0.5A]
//       Term 122 (EL2008) [EL2008 8Ch. Dig. Output 24V, 0.5A]
//       Term 123 (EL2008) [EL2008 8Ch. Dig. Output 24V, 0.5A]
//       Term 124 (EL2008) [EL2008 8Ch. Dig. Output 24V, 0.5A]
//       Term 111 (EL9011) [EL9011 End Terminal]
//     Drive PA10601 (ASDA-A2-E CoE Drive) [Delta ASDA-A2-E EtherCAT(CoE) Drive Rev4]
//     Drive PA10701 (ASDA-A2-E CoE Drive) [Delta ASDA-A2-E EtherCAT(CoE) Drive Rev4]
//     Drive PA10801 (ASDA-A2-E CoE Drive) [Delta ASDA-A2-E EtherCAT(CoE) Drive Rev4]
//     Drive PA10901 (ASDA-A2-E CoE Drive) [Delta ASDA-A2-E EtherCAT(CoE) Drive Rev4]
//     Drive PA11001 (ASDA-A2-E CoE Drive) [Delta ASDA-A2-E EtherCAT(CoE) Drive Rev4]
//   DEVICE Device 6 (NOV-DP-RAM)
//     Box 18 (Retain Handler)
// variable links:
//   NC-Task 1 SAF/Axes/Belt 1 <-> Device 4 (EtherCAT)/Drive PA12101 (ASDA-A2-E CoE Drive)
//     Drive/Inputs/In/nDataIn3[0] <-> 1st TxPDO Mapping/ActualTorque
//     Drive/Inputs/In/nDcOutputTime <-> InfoData/DcOutputShift
//     Drive/Inputs/In/nState1 <-> 1st TxPDO Mapping/Status Word
//     Drive/Inputs/In/nState2 <-> 1st TxPDO Mapping/Status Word @bit 8
//     Drive/Inputs/In/nState4 @bit 1 <-> WcState/InputToggle
//     Drive/Inputs/In/nState4 <-> WcState/WcState
//     Drive/Outputs/Out/nCtrl1 <-> 2nd RxPDO Mapping/Control Word
//     Drive/Outputs/Out/nCtrl2 <-> 2nd RxPDO Mapping/Control Word @bit 8
//     Drive/Outputs/Out/nDataOut1 <-> 2nd RxPDO Mapping/TargetPosition
//     Enc/Inputs/In/nDataIn1 <-> 1st TxPDO Mapping/ActualPosition
//     Enc/Inputs/In/nDataIn7 <-> 1st TxPDO Mapping/Velocity actual value
//     Enc/Inputs/In/nDcInputTime <-> InfoData/DcInputShift
//     Enc/Inputs/In/nState4 @bit 1 <-> WcState/InputToggle
//     Enc/Inputs/In/nState4 <-> WcState/WcState
//   NC-Task 1 SAF/Axes/Belt 2 <-> Device 4 (EtherCAT)/Drive PA13201 (ASDA-A2-E CoE Drive)
//     Drive/Inputs/In/nDataIn3[0] <-> 1st TxPDO Mapping/ActualTorque
//     Drive/Inputs/In/nDcOutputTime <-> InfoData/DcOutputShift
//     Drive/Inputs/In/nState1 <-> 1st TxPDO Mapping/Status Word
//     Drive/Inputs/In/nState2 <-> 1st TxPDO Mapping/Status Word @bit 8
//     Drive/Inputs/In/nState4 @bit 1 <-> WcState/InputToggle
//     Drive/Inputs/In/nState4 <-> WcState/WcState
//     Drive/Outputs/Out/nCtrl1 <-> 2nd RxPDO Mapping/Control Word
//     Drive/Outputs/Out/nCtrl2 <-> 2nd RxPDO Mapping/Control Word @bit 8
//     Drive/Outputs/Out/nDataOut1 <-> 2nd RxPDO Mapping/TargetPosition
//     Enc/Inputs/In/nDataIn1 <-> 1st TxPDO Mapping/ActualPosition
//     Enc/Inputs/In/nDataIn7 <-> 1st TxPDO Mapping/Velocity actual value
//     Enc/Inputs/In/nDcInputTime <-> InfoData/DcInputShift
//     Enc/Inputs/In/nState4 @bit 1 <-> WcState/InputToggle
//     Enc/Inputs/In/nState4 <-> WcState/WcState
//   NC-Task 1 SAF/Axes/Belt 3 <-> Device 4 (EtherCAT)/Drive PA14301 (ASDA-A2-E CoE Drive)
//     Drive/Inputs/In/nDataIn3[0] <-> 1st TxPDO Mapping/ActualTorque
//     Drive/Inputs/In/nDcOutputTime <-> InfoData/DcOutputShift
//     Drive/Inputs/In/nState1 <-> 1st TxPDO Mapping/Status Word
//     Drive/Inputs/In/nState2 <-> 1st TxPDO Mapping/Status Word @bit 8
//     Drive/Inputs/In/nState4 @bit 1 <-> WcState/InputToggle
//     Drive/Inputs/In/nState4 <-> WcState/WcState
//     Drive/Outputs/Out/nCtrl1 <-> 2nd RxPDO Mapping/Control Word
//     Drive/Outputs/Out/nCtrl2 <-> 2nd RxPDO Mapping/Control Word @bit 8
//     Drive/Outputs/Out/nDataOut1 <-> 2nd RxPDO Mapping/TargetPosition
//     Enc/Inputs/In/nDataIn1 <-> 1st TxPDO Mapping/ActualPosition
//     Enc/Inputs/In/nDataIn7 <-> 1st TxPDO Mapping/Velocity actual value
//     Enc/Inputs/In/nDcInputTime <-> InfoData/DcInputShift
//     Enc/Inputs/In/nState4 @bit 1 <-> WcState/InputToggle
//     Enc/Inputs/In/nState4 <-> WcState/WcState
//   NC-Task 1 SAF/Axes/Belt 4 <-> Device 1 (EtherCAT)/Term 1 (EK1200)/Term 17 (EK1122)/Drive PA14401 (ASDA-A2-E CoE Drive)
//     Drive/Inputs/In/nDataIn3[0] <-> 1st Transmit PDO Mapping/Torque actual value
//     Drive/Inputs/In/nDcOutputTime <-> InfoData/DcOutputShift
//     Drive/Inputs/In/nState1 <-> 1st Transmit PDO Mapping/Statusword
//     Drive/Inputs/In/nState2 <-> 1st Transmit PDO Mapping/Statusword @bit 8
//     Drive/Inputs/In/nState4 @bit 1 <-> WcState/InputToggle
//     Drive/Inputs/In/nState4 <-> WcState/WcState
//     Drive/Outputs/Out/nCtrl1 <-> 2nd Receive PDO Mapping/Controlword
//     Drive/Outputs/Out/nCtrl2 <-> 2nd Receive PDO Mapping/Controlword @bit 8
//     Drive/Outputs/Out/nDataOut1 <-> 2nd Receive PDO Mapping/Target position
//     Enc/Inputs/In/nDataIn1 <-> 1st Transmit PDO Mapping/Position actual value
//     Enc/Inputs/In/nDataIn7 <-> 1st Transmit PDO Mapping/Velocity actual value
//     Enc/Inputs/In/nDcInputTime <-> InfoData/DcInputShift
//     Enc/Inputs/In/nState4 @bit 1 <-> WcState/InputToggle
//     Enc/Inputs/In/nState4 <-> WcState/WcState
//   NC-Task 1 SAF/Axes/Belt 5 <-> Device 1 (EtherCAT)/Term 1 (EK1200)/Term 17 (EK1122)/Drive PA14501 (ASDA-A2-E CoE Drive)
//     Drive/Inputs/In/nDataIn3[0] <-> 1st Transmit PDO Mapping/Torque actual value
//     Drive/Inputs/In/nDcOutputTime <-> InfoData/DcOutputShift
//     Drive/Inputs/In/nState1 <-> 1st Transmit PDO Mapping/Statusword
//     Drive/Inputs/In/nState2 <-> 1st Transmit PDO Mapping/Statusword @bit 8
//     Drive/Inputs/In/nState4 @bit 1 <-> WcState/InputToggle
//     Drive/Inputs/In/nState4 <-> WcState/WcState
//     Drive/Outputs/Out/nCtrl1 <-> 2nd Receive PDO Mapping/Controlword
//     Drive/Outputs/Out/nCtrl2 <-> 2nd Receive PDO Mapping/Controlword @bit 8
//     Drive/Outputs/Out/nDataOut1 <-> 2nd Receive PDO Mapping/Target position
//     Enc/Inputs/In/nDataIn1 <-> 1st Transmit PDO Mapping/Position actual value
//     Enc/Inputs/In/nDataIn7 <-> 1st Transmit PDO Mapping/Velocity actual value
//     Enc/Inputs/In/nDcInputTime <-> InfoData/DcInputShift
//     Enc/Inputs/In/nState4 @bit 1 <-> WcState/InputToggle
//     Enc/Inputs/In/nState4 <-> WcState/WcState
//   NC-Task 1 SAF/Axes/Belt 6 <-> Device 1 (EtherCAT)/Term 1 (EK1200)/Term 17 (EK1122)/Drive PA14601 (ASDA-A2-E CoE Drive)
//     Drive/Inputs/In/nDataIn3[0] <-> 1st TxPDO Mapping/ActualTorque
//     Drive/Inputs/In/nDcOutputTime <-> InfoData/DcOutputShift
//     Drive/Inputs/In/nState1 <-> 1st TxPDO Mapping/Status Word
//     Drive/Inputs/In/nState2 <-> 1st TxPDO Mapping/Status Word @bit 8
//     Drive/Inputs/In/nState4 @bit 1 <-> WcState/InputToggle
//     Drive/Inputs/In/nState4 <-> WcState/WcState
//     Drive/Outputs/Out/nCtrl1 <-> 2nd RxPDO Mapping/Control Word
//     Drive/Outputs/Out/nCtrl2 <-> 2nd RxPDO Mapping/Control Word @bit 8
//     Drive/Outputs/Out/nDataOut1 <-> 2nd RxPDO Mapping/TargetPosition
//     Enc/Inputs/In/nDataIn1 <-> 1st TxPDO Mapping/ActualPosition
//     Enc/Inputs/In/nDataIn7 <-> 1st TxPDO Mapping/Velocity actual value
//     Enc/Inputs/In/nDcInputTime <-> InfoData/DcInputShift
//     Enc/Inputs/In/nState4 @bit 1 <-> WcState/InputToggle
//     Enc/Inputs/In/nState4 <-> WcState/WcState
//   NC-Task 1 SAF/Axes/Belt7 <-> Device 1 (EtherCAT)/Drive PA14901 (ASDA-A2-E CoE Drive)
//     Drive/Inputs/In/nDataIn3[0] <-> 1st TxPDO Mapping/ActualTorque
//     Drive/Inputs/In/nDcOutputTime <-> InfoData/DcOutputShift
//     Drive/Inputs/In/nState1 <-> 1st TxPDO Mapping/Status Word
//     Drive/Inputs/In/nState2 <-> 1st TxPDO Mapping/Status Word @bit 8
//     Drive/Inputs/In/nState4 @bit 1 <-> WcState/InputToggle
//     Drive/Inputs/In/nState4 <-> WcState/WcState
//     Drive/Outputs/Out/nCtrl1 <-> 2nd RxPDO Mapping/Control Word
//     Drive/Outputs/Out/nCtrl2 <-> 2nd RxPDO Mapping/Control Word @bit 8
//     Drive/Outputs/Out/nDataOut1 <-> 2nd RxPDO Mapping/TargetPosition
//     Enc/Inputs/In/nDataIn1 <-> 1st TxPDO Mapping/ActualPosition
//     Enc/Inputs/In/nDataIn7 <-> 1st TxPDO Mapping/Velocity actual value
//     Enc/Inputs/In/nDcInputTime <-> InfoData/DcInputShift
//     Enc/Inputs/In/nState4 @bit 1 <-> WcState/InputToggle
//     Enc/Inputs/In/nState4 <-> WcState/WcState
//   NC-Task 1 SAF/Axes/Counter 1 <-> Device 4 (EtherCAT)/Drive PA10101 (ASDA-A2-E CoE Drive)
//     Drive/Inputs/In/nDataIn3[0] <-> 1st TxPDO Mapping/ActualTorque
//     Drive/Inputs/In/nDcOutputTime <-> InfoData/DcOutputShift
//     Drive/Inputs/In/nState1 <-> 1st TxPDO Mapping/Status Word
//     Drive/Inputs/In/nState2 <-> 1st TxPDO Mapping/Status Word @bit 8
//     Drive/Inputs/In/nState4 @bit 1 <-> WcState/InputToggle
//     Drive/Inputs/In/nState4 <-> WcState/WcState
//     Drive/Outputs/Out/nCtrl1 <-> 2nd RxPDO Mapping/Control Word
//     Drive/Outputs/Out/nCtrl2 <-> 2nd RxPDO Mapping/Control Word @bit 8
//     Drive/Outputs/Out/nDataOut1 <-> 2nd RxPDO Mapping/TargetPosition
//     Enc/Inputs/In/nDataIn1 <-> 1st TxPDO Mapping/ActualPosition
//     Enc/Inputs/In/nDataIn7 <-> 1st TxPDO Mapping/Velocity actual value
//     Enc/Inputs/In/nDcInputTime <-> InfoData/DcInputShift
//     Enc/Inputs/In/nState4 @bit 1 <-> WcState/InputToggle
//     Enc/Inputs/In/nState4 <-> WcState/WcState
//   NC-Task 1 SAF/Axes/Counter 10 <-> Device 4 (EtherCAT)/Drive PA11001 (ASDA-A2-E CoE Drive)
//     Drive/Inputs/In/nDataIn3[0] <-> 1st TxPDO Mapping/ActualTorque
//     Drive/Inputs/In/nDcOutputTime <-> InfoData/DcOutputShift
//     Drive/Inputs/In/nState1 <-> 1st TxPDO Mapping/Status Word
//     Drive/Inputs/In/nState2 <-> 1st TxPDO Mapping/Status Word @bit 8
//     Drive/Inputs/In/nState4 @bit 1 <-> WcState/InputToggle
//     Drive/Inputs/In/nState4 <-> WcState/WcState
//     Drive/Outputs/Out/nCtrl1 <-> 2nd RxPDO Mapping/Control Word
//     Drive/Outputs/Out/nCtrl2 <-> 2nd RxPDO Mapping/Control Word @bit 8
//     Drive/Outputs/Out/nDataOut1 <-> 2nd RxPDO Mapping/TargetPosition
//     Enc/Inputs/In/nDataIn1 <-> 1st TxPDO Mapping/ActualPosition
//     Enc/Inputs/In/nDataIn7 <-> 1st TxPDO Mapping/Velocity actual value
//     Enc/Inputs/In/nDcInputTime <-> InfoData/DcInputShift
//     Enc/Inputs/In/nState4 @bit 1 <-> WcState/InputToggle
//     Enc/Inputs/In/nState4 <-> WcState/WcState
//   NC-Task 1 SAF/Axes/Counter 11 <-> Device 4 (EtherCAT)/Drive PA11101 (ASDA-A2-E CoE Drive)
//     Drive/Inputs/In/nDataIn3[0] <-> 1st TxPDO Mapping/ActualTorque
//     Drive/Inputs/In/nDcOutputTime <-> InfoData/DcOutputShift
//     Drive/Inputs/In/nState1 <-> 1st TxPDO Mapping/Status Word
//     Drive/Inputs/In/nState2 <-> 1st TxPDO Mapping/Status Word @bit 8
//     Drive/Inputs/In/nState4 @bit 1 <-> WcState/InputToggle
//     Drive/Inputs/In/nState4 <-> WcState/WcState
//     Drive/Outputs/Out/nCtrl1 <-> 2nd RxPDO Mapping/Control Word
//     Drive/Outputs/Out/nCtrl2 <-> 2nd RxPDO Mapping/Control Word @bit 8
//     Drive/Outputs/Out/nDataOut1 <-> 2nd RxPDO Mapping/TargetPosition
//     Enc/Inputs/In/nDataIn1 <-> 1st TxPDO Mapping/ActualPosition
//     Enc/Inputs/In/nDataIn7 <-> 1st TxPDO Mapping/Velocity actual value
//     Enc/Inputs/In/nDcInputTime <-> InfoData/DcInputShift
//     Enc/Inputs/In/nState4 @bit 1 <-> WcState/InputToggle
//     Enc/Inputs/In/nState4 <-> WcState/WcState
//   NC-Task 1 SAF/Axes/Counter 12 <-> Device 4 (EtherCAT)/Drive PA11201 (ASDA-A2-E CoE Drive)
//     Drive/Inputs/In/nDataIn3[0] <-> 1st TxPDO Mapping/ActualTorque
//     Drive/Inputs/In/nDcOutputTime <-> InfoData/DcOutputShift
//     Drive/Inputs/In/nState1 <-> 1st TxPDO Mapping/Status Word
//     Drive/Inputs/In/nState2 <-> 1st TxPDO Mapping/Status Word @bit 8
//     Drive/Inputs/In/nState4 @bit 1 <-> WcState/InputToggle
//     Drive/Inputs/In/nState4 <-> WcState/WcState
//     Drive/Outputs/Out/nCtrl1 <-> 2nd RxPDO Mapping/Control Word
//     Drive/Outputs/Out/nCtrl2 <-> 2nd RxPDO Mapping/Control Word @bit 8
//     Drive/Outputs/Out/nDataOut1 <-> 2nd RxPDO Mapping/TargetPosition
//     Enc/Inputs/In/nDataIn1 <-> 1st TxPDO Mapping/ActualPosition
//     Enc/Inputs/In/nDataIn7 <-> 1st TxPDO Mapping/Velocity actual value
//     Enc/Inputs/In/nDcInputTime <-> InfoData/DcInputShift
//     Enc/Inputs/In/nState4 @bit 1 <-> WcState/InputToggle
//     Enc/Inputs/In/nState4 <-> WcState/WcState
//   NC-Task 1 SAF/Axes/Counter 13 <-> Device 4 (EtherCAT)/Drive PA11301 (ASDA-A2-E CoE Drive)
//     Drive/Inputs/In/nDataIn3[0] <-> 1st TxPDO Mapping/ActualTorque
//     Drive/Inputs/In/nDcOutputTime <-> InfoData/DcOutputShift
//     Drive/Inputs/In/nState1 <-> 1st TxPDO Mapping/Status Word
//     Drive/Inputs/In/nState2 <-> 1st TxPDO Mapping/Status Word @bit 8
//     Drive/Inputs/In/nState4 @bit 1 <-> WcState/InputToggle
//     Drive/Inputs/In/nState4 <-> WcState/WcState
//     Drive/Outputs/Out/nCtrl1 <-> 2nd RxPDO Mapping/Control Word
//     Drive/Outputs/Out/nCtrl2 <-> 2nd RxPDO Mapping/Control Word @bit 8
//     Drive/Outputs/Out/nDataOut1 <-> 2nd RxPDO Mapping/TargetPosition
//     Enc/Inputs/In/nDataIn1 <-> 1st TxPDO Mapping/ActualPosition
//     Enc/Inputs/In/nDataIn7 <-> 1st TxPDO Mapping/Velocity actual value
//     Enc/Inputs/In/nDcInputTime <-> InfoData/DcInputShift
//     Enc/Inputs/In/nState4 @bit 1 <-> WcState/InputToggle
//     Enc/Inputs/In/nState4 <-> WcState/WcState
//   NC-Task 1 SAF/Axes/Counter 14 <-> Device 4 (EtherCAT)/Drive PA11401 (ASDA-A2-E CoE Drive)
//     Drive/Inputs/In/nDataIn3[0] <-> 1st TxPDO Mapping/ActualTorque
//     Drive/Inputs/In/nDcOutputTime <-> InfoData/DcOutputShift
//     Drive/Inputs/In/nState1 <-> 1st TxPDO Mapping/Status Word
//     Drive/Inputs/In/nState2 <-> 1st TxPDO Mapping/Status Word @bit 8
//     Drive/Inputs/In/nState4 @bit 1 <-> WcState/InputToggle
//     Drive/Inputs/In/nState4 <-> WcState/WcState
//     Drive/Outputs/Out/nCtrl1 <-> 2nd RxPDO Mapping/Control Word
//     Drive/Outputs/Out/nCtrl2 <-> 2nd RxPDO Mapping/Control Word @bit 8
//     Drive/Outputs/Out/nDataOut1 <-> 2nd RxPDO Mapping/TargetPosition
//     Enc/Inputs/In/nDataIn1 <-> 1st TxPDO Mapping/ActualPosition
//     Enc/Inputs/In/nDataIn7 <-> 1st TxPDO Mapping/Velocity actual value
//     Enc/Inputs/In/nDcInputTime <-> InfoData/DcInputShift
//     Enc/Inputs/In/nState4 @bit 1 <-> WcState/InputToggle
//     Enc/Inputs/In/nState4 <-> WcState/WcState
//   NC-Task 1 SAF/Axes/Counter 15 <-> Device 4 (EtherCAT)/Drive PA11501 (ASDA-A2-E CoE Drive)
//     Drive/Inputs/In/nDataIn3[0] <-> 1st TxPDO Mapping/ActualTorque
//     Drive/Inputs/In/nDcOutputTime <-> InfoData/DcOutputShift
//     Drive/Inputs/In/nState1 <-> 1st TxPDO Mapping/Status Word
//     Drive/Inputs/In/nState2 <-> 1st TxPDO Mapping/Status Word @bit 8
//     Drive/Inputs/In/nState4 @bit 1 <-> WcState/InputToggle
//     Drive/Inputs/In/nState4 <-> WcState/WcState
//     Drive/Outputs/Out/nCtrl1 <-> 2nd RxPDO Mapping/Control Word
//     Drive/Outputs/Out/nCtrl2 <-> 2nd RxPDO Mapping/Control Word @bit 8
//     Drive/Outputs/Out/nDataOut1 <-> 2nd RxPDO Mapping/TargetPosition
//     Enc/Inputs/In/nDataIn1 <-> 1st TxPDO Mapping/ActualPosition
//     Enc/Inputs/In/nDataIn7 <-> 1st TxPDO Mapping/Velocity actual value
//     Enc/Inputs/In/nDcInputTime <-> InfoData/DcInputShift
//     Enc/Inputs/In/nState4 @bit 1 <-> WcState/InputToggle
//     Enc/Inputs/In/nState4 <-> WcState/WcState
//   NC-Task 1 SAF/Axes/Counter 16 <-> Device 4 (EtherCAT)/Drive PA11601 (ASDA-A2-E CoE Drive)
//     Drive/Inputs/In/nDataIn3[0] <-> 1st TxPDO Mapping/ActualTorque
//     Drive/Inputs/In/nDcOutputTime <-> InfoData/DcOutputShift
//     Drive/Inputs/In/nState1 <-> 1st TxPDO Mapping/Status Word
//     Drive/Inputs/In/nState2 <-> 1st TxPDO Mapping/Status Word @bit 8
//     Drive/Inputs/In/nState4 @bit 1 <-> WcState/InputToggle
//     Drive/Inputs/In/nState4 <-> WcState/WcState
//     Drive/Outputs/Out/nCtrl1 <-> 2nd RxPDO Mapping/Control Word
//     Drive/Outputs/Out/nCtrl2 <-> 2nd RxPDO Mapping/Control Word @bit 8
//     Drive/Outputs/Out/nDataOut1 <-> 2nd RxPDO Mapping/TargetPosition
//     Enc/Inputs/In/nDataIn1 <-> 1st TxPDO Mapping/ActualPosition
//     Enc/Inputs/In/nDataIn7 <-> 1st TxPDO Mapping/Velocity actual value
//     Enc/Inputs/In/nDcInputTime <-> InfoData/DcInputShift
//     Enc/Inputs/In/nState4 @bit 1 <-> WcState/InputToggle
//     Enc/Inputs/In/nState4 <-> WcState/WcState
//   NC-Task 1 SAF/Axes/Counter 17 <-> Device 4 (EtherCAT)/Drive PA11701 (ASDA-A2-E CoE Drive)
//     Drive/Inputs/In/nDataIn3[0] <-> 1st TxPDO Mapping/ActualTorque
//     Drive/Inputs/In/nDcOutputTime <-> InfoData/DcOutputShift
//     Drive/Inputs/In/nState1 <-> 1st TxPDO Mapping/Status Word
//     Drive/Inputs/In/nState2 <-> 1st TxPDO Mapping/Status Word @bit 8
//     Drive/Inputs/In/nState4 @bit 1 <-> WcState/InputToggle
//     Drive/Inputs/In/nState4 <-> WcState/WcState
//     Drive/Outputs/Out/nCtrl1 <-> 2nd RxPDO Mapping/Control Word
//     Drive/Outputs/Out/nCtrl2 <-> 2nd RxPDO Mapping/Control Word @bit 8
//     Drive/Outputs/Out/nDataOut1 <-> 2nd RxPDO Mapping/TargetPosition
//     Enc/Inputs/In/nDataIn1 <-> 1st TxPDO Mapping/ActualPosition
//     Enc/Inputs/In/nDataIn7 <-> 1st TxPDO Mapping/Velocity actual value
//     Enc/Inputs/In/nDcInputTime <-> InfoData/DcInputShift
//     Enc/Inputs/In/nState4 @bit 1 <-> WcState/InputToggle
//     Enc/Inputs/In/nState4 <-> WcState/WcState
//   NC-Task 1 SAF/Axes/Counter 18 <-> Device 4 (EtherCAT)/Drive PA11801 (ASDA-A2-E CoE Drive)
//     Drive/Inputs/In/nDataIn3[0] <-> 1st TxPDO Mapping/ActualTorque
//     Drive/Inputs/In/nDcOutputTime <-> InfoData/DcOutputShift
//     Drive/Inputs/In/nState1 <-> 1st TxPDO Mapping/Status Word
//     Drive/Inputs/In/nState2 <-> 1st TxPDO Mapping/Status Word @bit 8
//     Drive/Inputs/In/nState4 @bit 1 <-> WcState/InputToggle
//     Drive/Inputs/In/nState4 <-> WcState/WcState
//     Drive/Outputs/Out/nCtrl1 <-> 2nd RxPDO Mapping/Control Word
//     Drive/Outputs/Out/nCtrl2 <-> 2nd RxPDO Mapping/Control Word @bit 8
//     Drive/Outputs/Out/nDataOut1 <-> 2nd RxPDO Mapping/TargetPosition
//     Enc/Inputs/In/nDataIn1 <-> 1st TxPDO Mapping/ActualPosition
//     Enc/Inputs/In/nDataIn7 <-> 1st TxPDO Mapping/Velocity actual value
//     Enc/Inputs/In/nDcInputTime <-> InfoData/DcInputShift
//     Enc/Inputs/In/nState4 @bit 1 <-> WcState/InputToggle
//     Enc/Inputs/In/nState4 <-> WcState/WcState
//   NC-Task 1 SAF/Axes/Counter 19 <-> Device 4 (EtherCAT)/Drive PA11901 (ASDA-A2-E CoE Drive)
//     Drive/Inputs/In/nDataIn3[0] <-> 1st TxPDO Mapping/ActualTorque
//     Drive/Inputs/In/nDcOutputTime <-> InfoData/DcOutputShift
//     Drive/Inputs/In/nState1 <-> 1st TxPDO Mapping/Status Word
//     Drive/Inputs/In/nState2 <-> 1st TxPDO Mapping/Status Word @bit 8
//     Drive/Inputs/In/nState4 @bit 1 <-> WcState/InputToggle
//     Drive/Inputs/In/nState4 <-> WcState/WcState
//     Drive/Outputs/Out/nCtrl1 <-> 2nd RxPDO Mapping/Control Word
//     Drive/Outputs/Out/nCtrl2 <-> 2nd RxPDO Mapping/Control Word @bit 8
//     Drive/Outputs/Out/nDataOut1 <-> 2nd RxPDO Mapping/TargetPosition
//     Enc/Inputs/In/nDataIn1 <-> 1st TxPDO Mapping/ActualPosition
//     Enc/Inputs/In/nDataIn7 <-> 1st TxPDO Mapping/Velocity actual value
//     Enc/Inputs/In/nDcInputTime <-> InfoData/DcInputShift
//     Enc/Inputs/In/nState4 @bit 1 <-> WcState/InputToggle
//     Enc/Inputs/In/nState4 <-> WcState/WcState
//   NC-Task 1 SAF/Axes/Counter 2 <-> Device 4 (EtherCAT)/Drive PA10201 (ASDA-A2-E CoE Drive)
//     Drive/Inputs/In/nDataIn3[0] <-> 1st TxPDO Mapping/ActualTorque
//     Drive/Inputs/In/nDcOutputTime <-> InfoData/DcOutputShift
//     Drive/Inputs/In/nState1 <-> 1st TxPDO Mapping/Status Word
//     Drive/Inputs/In/nState2 <-> 1st TxPDO Mapping/Status Word @bit 8
//     Drive/Inputs/In/nState4 @bit 1 <-> WcState/InputToggle
//     Drive/Inputs/In/nState4 <-> WcState/WcState
//     Drive/Outputs/Out/nCtrl1 <-> 2nd RxPDO Mapping/Control Word
//     Drive/Outputs/Out/nCtrl2 <-> 2nd RxPDO Mapping/Control Word @bit 8
//     Drive/Outputs/Out/nDataOut1 <-> 2nd RxPDO Mapping/TargetPosition
//     Enc/Inputs/In/nDataIn1 <-> 1st TxPDO Mapping/ActualPosition
//     Enc/Inputs/In/nDataIn7 <-> 1st TxPDO Mapping/Velocity actual value
//     Enc/Inputs/In/nDcInputTime <-> InfoData/DcInputShift
//     Enc/Inputs/In/nState4 @bit 1 <-> WcState/InputToggle
//     Enc/Inputs/In/nState4 <-> WcState/WcState
//   NC-Task 1 SAF/Axes/Counter 20 <-> Device 4 (EtherCAT)/Drive PA12001 (ASDA-A2-E CoE Drive)
//     Drive/Inputs/In/nDataIn3[0] <-> 1st TxPDO Mapping/ActualTorque
//     Drive/Inputs/In/nDcOutputTime <-> InfoData/DcOutputShift
//     Drive/Inputs/In/nState1 <-> 1st TxPDO Mapping/Status Word
//     Drive/Inputs/In/nState2 <-> 1st TxPDO Mapping/Status Word @bit 8
//     Drive/Inputs/In/nState4 @bit 1 <-> WcState/InputToggle
//     Drive/Inputs/In/nState4 <-> WcState/WcState
//     Drive/Outputs/Out/nCtrl1 <-> 2nd RxPDO Mapping/Control Word
//     Drive/Outputs/Out/nCtrl2 <-> 2nd RxPDO Mapping/Control Word @bit 8
//     Drive/Outputs/Out/nDataOut1 <-> 2nd RxPDO Mapping/TargetPosition
//     Enc/Inputs/In/nDataIn1 <-> 1st TxPDO Mapping/ActualPosition
//     Enc/Inputs/In/nDataIn7 <-> 1st TxPDO Mapping/Velocity actual value
//     Enc/Inputs/In/nDcInputTime <-> InfoData/DcInputShift
//     Enc/Inputs/In/nState4 @bit 1 <-> WcState/InputToggle
//     Enc/Inputs/In/nState4 <-> WcState/WcState
//   NC-Task 1 SAF/Axes/Counter 21 <-> Device 4 (EtherCAT)/Drive PA12201 (ASDA-A2-E CoE Drive)
//     Drive/Inputs/In/nDataIn3[0] <-> 1st TxPDO Mapping/ActualTorque
//     Drive/Inputs/In/nDcOutputTime <-> InfoData/DcOutputShift
//     Drive/Inputs/In/nState1 <-> 1st TxPDO Mapping/Status Word
//     Drive/Inputs/In/nState2 <-> 1st TxPDO Mapping/Status Word @bit 8
//     Drive/Inputs/In/nState4 @bit 1 <-> WcState/InputToggle
//     Drive/Inputs/In/nState4 <-> WcState/WcState
//     Drive/Outputs/Out/nCtrl1 <-> 2nd RxPDO Mapping/Control Word
//     Drive/Outputs/Out/nCtrl2 <-> 2nd RxPDO Mapping/Control Word @bit 8
//     Drive/Outputs/Out/nDataOut1 <-> 2nd RxPDO Mapping/TargetPosition
//     Enc/Inputs/In/nDataIn1 <-> 1st TxPDO Mapping/ActualPosition
//     Enc/Inputs/In/nDataIn7 <-> 1st TxPDO Mapping/Velocity actual value
//     Enc/Inputs/In/nDcInputTime <-> InfoData/DcInputShift
//     Enc/Inputs/In/nState4 @bit 1 <-> WcState/InputToggle
//     Enc/Inputs/In/nState4 <-> WcState/WcState
//   NC-Task 1 SAF/Axes/Counter 22 <-> Device 4 (EtherCAT)/Drive PA12301 (ASDA-A2-E CoE Drive)
//     Drive/Inputs/In/nDataIn3[0] <-> 1st TxPDO Mapping/ActualTorque
//     Drive/Inputs/In/nDcOutputTime <-> InfoData/DcOutputShift
//     Drive/Inputs/In/nState1 <-> 1st TxPDO Mapping/Status Word
//     Drive/Inputs/In/nState2 <-> 1st TxPDO Mapping/Status Word @bit 8
//     Drive/Inputs/In/nState4 @bit 1 <-> WcState/InputToggle
//     Drive/Inputs/In/nState4 <-> WcState/WcState
//     Drive/Outputs/Out/nCtrl1 <-> 2nd RxPDO Mapping/Control Word
//     Drive/Outputs/Out/nCtrl2 <-> 2nd RxPDO Mapping/Control Word @bit 8
//     Drive/Outputs/Out/nDataOut1 <-> 2nd RxPDO Mapping/TargetPosition
//     Enc/Inputs/In/nDataIn1 <-> 1st TxPDO Mapping/ActualPosition
//     Enc/Inputs/In/nDataIn7 <-> 1st TxPDO Mapping/Velocity actual value
//     Enc/Inputs/In/nDcInputTime <-> InfoData/DcInputShift
//     Enc/Inputs/In/nState4 @bit 1 <-> WcState/InputToggle
//     Enc/Inputs/In/nState4 <-> WcState/WcState
//   NC-Task 1 SAF/Axes/Counter 23 <-> Device 4 (EtherCAT)/Drive PA12401 (ASDA-A2-E CoE Drive)
//     Drive/Inputs/In/nDataIn3[0] <-> 1st TxPDO Mapping/ActualTorque
//     Drive/Inputs/In/nDcOutputTime <-> InfoData/DcOutputShift
//     Drive/Inputs/In/nState1 <-> 1st TxPDO Mapping/Status Word
//     Drive/Inputs/In/nState2 <-> 1st TxPDO Mapping/Status Word @bit 8
//     Drive/Inputs/In/nState4 @bit 1 <-> WcState/InputToggle
//     Drive/Inputs/In/nState4 <-> WcState/WcState
//     Drive/Outputs/Out/nCtrl1 <-> 2nd RxPDO Mapping/Control Word
//     Drive/Outputs/Out/nCtrl2 <-> 2nd RxPDO Mapping/Control Word @bit 8
//     Drive/Outputs/Out/nDataOut1 <-> 2nd RxPDO Mapping/TargetPosition
//     Enc/Inputs/In/nDataIn1 <-> 1st TxPDO Mapping/ActualPosition
//     Enc/Inputs/In/nDataIn7 <-> 1st TxPDO Mapping/Velocity actual value
//     Enc/Inputs/In/nDcInputTime <-> InfoData/DcInputShift
//     Enc/Inputs/In/nState4 @bit 1 <-> WcState/InputToggle
//     Enc/Inputs/In/nState4 <-> WcState/WcState
//   NC-Task 1 SAF/Axes/Counter 24 <-> Device 4 (EtherCAT)/Drive PA12501 (ASDA-A2-E CoE Drive)
//     Drive/Inputs/In/nDataIn3[0] <-> 1st TxPDO Mapping/ActualTorque
//     Drive/Inputs/In/nDcOutputTime <-> InfoData/DcOutputShift
//     Drive/Inputs/In/nState1 <-> 1st TxPDO Mapping/Status Word
//     Drive/Inputs/In/nState2 <-> 1st TxPDO Mapping/Status Word @bit 8
//     Drive/Inputs/In/nState4 @bit 1 <-> WcState/InputToggle
//     Drive/Inputs/In/nState4 <-> WcState/WcState
//     Drive/Outputs/Out/nCtrl1 <-> 2nd RxPDO Mapping/Control Word
//     Drive/Outputs/Out/nCtrl2 <-> 2nd RxPDO Mapping/Control Word @bit 8
//     Drive/Outputs/Out/nDataOut1 <-> 2nd RxPDO Mapping/TargetPosition
//     Enc/Inputs/In/nDataIn1 <-> 1st TxPDO Mapping/ActualPosition
//     Enc/Inputs/In/nDataIn7 <-> 1st TxPDO Mapping/Velocity actual value
//     Enc/Inputs/In/nDcInputTime <-> InfoData/DcInputShift
//     Enc/Inputs/In/nState4 @bit 1 <-> WcState/InputToggle
//     Enc/Inputs/In/nState4 <-> WcState/WcState
//   NC-Task 1 SAF/Axes/Counter 25 <-> Device 4 (EtherCAT)/Drive PA12601 (ASDA-A2-E CoE Drive)
//     Drive/Inputs/In/nDataIn3[0] <-> 1st TxPDO Mapping/ActualTorque
//     Drive/Inputs/In/nDcOutputTime <-> InfoData/DcOutputShift
//     Drive/Inputs/In/nState1 <-> 1st TxPDO Mapping/Status Word
//     Drive/Inputs/In/nState2 <-> 1st TxPDO Mapping/Status Word @bit 8
//     Drive/Inputs/In/nState4 @bit 1 <-> WcState/InputToggle
//     Drive/Inputs/In/nState4 <-> WcState/WcState
//     Drive/Outputs/Out/nCtrl1 <-> 2nd RxPDO Mapping/Control Word
//     Drive/Outputs/Out/nCtrl2 <-> 2nd RxPDO Mapping/Control Word @bit 8
//     Drive/Outputs/Out/nDataOut1 <-> 2nd RxPDO Mapping/TargetPosition
//     Enc/Inputs/In/nDataIn1 <-> 1st TxPDO Mapping/ActualPosition
//     Enc/Inputs/In/nDataIn7 <-> 1st TxPDO Mapping/Velocity actual value
//     Enc/Inputs/In/nDcInputTime <-> InfoData/DcInputShift
//     Enc/Inputs/In/nState4 @bit 1 <-> WcState/InputToggle
//     Enc/Inputs/In/nState4 <-> WcState/WcState
//   NC-Task 1 SAF/Axes/Counter 26 <-> Device 4 (EtherCAT)/Drive PA12701 (ASDA-A2-E CoE Drive)
//     Drive/Inputs/In/nDataIn3[0] <-> 1st TxPDO Mapping/ActualTorque
//     Drive/Inputs/In/nDcOutputTime <-> InfoData/DcOutputShift
//     Drive/Inputs/In/nState1 <-> 1st TxPDO Mapping/Status Word
//     Drive/Inputs/In/nState2 <-> 1st TxPDO Mapping/Status Word @bit 8
//     Drive/Inputs/In/nState4 @bit 1 <-> WcState/InputToggle
//     Drive/Inputs/In/nState4 <-> WcState/WcState
//     Drive/Outputs/Out/nCtrl1 <-> 2nd RxPDO Mapping/Control Word
//     Drive/Outputs/Out/nCtrl2 <-> 2nd RxPDO Mapping/Control Word @bit 8
//     Drive/Outputs/Out/nDataOut1 <-> 2nd RxPDO Mapping/TargetPosition
//     Enc/Inputs/In/nDataIn1 <-> 1st TxPDO Mapping/ActualPosition
//     Enc/Inputs/In/nDataIn7 <-> 1st TxPDO Mapping/Velocity actual value
//     Enc/Inputs/In/nDcInputTime <-> InfoData/DcInputShift
//     Enc/Inputs/In/nState4 @bit 1 <-> WcState/InputToggle
//     Enc/Inputs/In/nState4 <-> WcState/WcState
//   NC-Task 1 SAF/Axes/Counter 27 <-> Device 4 (EtherCAT)/Drive PA12801 (ASDA-A2-E CoE Drive)
//     Drive/Inputs/In/nDataIn3[0] <-> 1st TxPDO Mapping/ActualTorque
//     Drive/Inputs/In/nDcOutputTime <-> InfoData/DcOutputShift
//     Drive/Inputs/In/nState1 <-> 1st TxPDO Mapping/Status Word
//     Drive/Inputs/In/nState2 <-> 1st TxPDO Mapping/Status Word @bit 8
//     Drive/Inputs/In/nState4 @bit 1 <-> WcState/InputToggle
//     Drive/Inputs/In/nState4 <-> WcState/WcState
//     Drive/Outputs/Out/nCtrl1 <-> 2nd RxPDO Mapping/Control Word
//     Drive/Outputs/Out/nCtrl2 <-> 2nd RxPDO Mapping/Control Word @bit 8
//     Drive/Outputs/Out/nDataOut1 <-> 2nd RxPDO Mapping/TargetPosition
//     Enc/Inputs/In/nDataIn1 <-> 1st TxPDO Mapping/ActualPosition
//     Enc/Inputs/In/nDataIn7 <-> 1st TxPDO Mapping/Velocity actual value
//     Enc/Inputs/In/nDcInputTime <-> InfoData/DcInputShift
//     Enc/Inputs/In/nState4 @bit 1 <-> WcState/InputToggle
//     Enc/Inputs/In/nState4 <-> WcState/WcState
//   NC-Task 1 SAF/Axes/Counter 28 <-> Device 4 (EtherCAT)/Drive PA12901 (ASDA-A2-E CoE Drive)
//     Drive/Inputs/In/nDataIn3[0] <-> 1st TxPDO Mapping/ActualTorque
//     Drive/Inputs/In/nDcOutputTime <-> InfoData/DcOutputShift
//     Drive/Inputs/In/nState1 <-> 1st TxPDO Mapping/Status Word
//     Drive/Inputs/In/nState2 <-> 1st TxPDO Mapping/Status Word @bit 8
//     Drive/Inputs/In/nState4 @bit 1 <-> WcState/InputToggle
//     Drive/Inputs/In/nState4 <-> WcState/WcState
//     Drive/Outputs/Out/nCtrl1 <-> 2nd RxPDO Mapping/Control Word
//     Drive/Outputs/Out/nCtrl2 <-> 2nd RxPDO Mapping/Control Word @bit 8
//     Drive/Outputs/Out/nDataOut1 <-> 2nd RxPDO Mapping/TargetPosition
//     Enc/Inputs/In/nDataIn1 <-> 1st TxPDO Mapping/ActualPosition
//     Enc/Inputs/In/nDataIn7 <-> 1st TxPDO Mapping/Velocity actual value
//     Enc/Inputs/In/nDcInputTime <-> InfoData/DcInputShift
//     Enc/Inputs/In/nState4 @bit 1 <-> WcState/InputToggle
//     Enc/Inputs/In/nState4 <-> WcState/WcState
//   NC-Task 1 SAF/Axes/Counter 29 <-> Device 4 (EtherCAT)/Drive PA13001 (ASDA-A2-E CoE Drive)
//     Drive/Inputs/In/nDataIn3[0] <-> 1st TxPDO Mapping/ActualTorque
//     Drive/Inputs/In/nDcOutputTime <-> InfoData/DcOutputShift
//     Drive/Inputs/In/nState1 <-> 1st TxPDO Mapping/Status Word
//     Drive/Inputs/In/nState2 <-> 1st TxPDO Mapping/Status Word @bit 8
//     Drive/Inputs/In/nState4 @bit 1 <-> WcState/InputToggle
//     Drive/Inputs/In/nState4 <-> WcState/WcState
//     Drive/Outputs/Out/nCtrl1 <-> 2nd RxPDO Mapping/Control Word
//     Drive/Outputs/Out/nCtrl2 <-> 2nd RxPDO Mapping/Control Word @bit 8
//     Drive/Outputs/Out/nDataOut1 <-> 2nd RxPDO Mapping/TargetPosition
//     Enc/Inputs/In/nDataIn1 <-> 1st TxPDO Mapping/ActualPosition
//     Enc/Inputs/In/nDataIn7 <-> 1st TxPDO Mapping/Velocity actual value
//     Enc/Inputs/In/nDcInputTime <-> InfoData/DcInputShift
//     Enc/Inputs/In/nState4 @bit 1 <-> WcState/InputToggle
//     Enc/Inputs/In/nState4 <-> WcState/WcState
//   NC-Task 1 SAF/Axes/Counter 3 <-> Device 4 (EtherCAT)/Drive PA10301 (ASDA-A2-E CoE Drive)
//     Drive/Inputs/In/nDataIn3[0] <-> 1st TxPDO Mapping/ActualTorque
//     Drive/Inputs/In/nDcOutputTime <-> InfoData/DcOutputShift
//     Drive/Inputs/In/nState1 <-> 1st TxPDO Mapping/Status Word
//     Drive/Inputs/In/nState2 <-> 1st TxPDO Mapping/Status Word @bit 8
//     Drive/Inputs/In/nState4 @bit 1 <-> WcState/InputToggle
//     Drive/Inputs/In/nState4 <-> WcState/WcState
//     Drive/Outputs/Out/nCtrl1 <-> 2nd RxPDO Mapping/Control Word
//     Drive/Outputs/Out/nCtrl2 <-> 2nd RxPDO Mapping/Control Word @bit 8
//     Drive/Outputs/Out/nDataOut1 <-> 2nd RxPDO Mapping/TargetPosition
//     Enc/Inputs/In/nDataIn1 <-> 1st TxPDO Mapping/ActualPosition
//     Enc/Inputs/In/nDataIn7 <-> 1st TxPDO Mapping/Velocity actual value
//     Enc/Inputs/In/nDcInputTime <-> InfoData/DcInputShift
//     Enc/Inputs/In/nState4 @bit 1 <-> WcState/InputToggle
//     Enc/Inputs/In/nState4 <-> WcState/WcState
//   NC-Task 1 SAF/Axes/Counter 30 <-> Device 4 (EtherCAT)/Drive PA13101 (ASDA-A2-E CoE Drive)
//     Drive/Inputs/In/nDataIn3[0] <-> 1st TxPDO Mapping/ActualTorque
//     Drive/Inputs/In/nDcOutputTime <-> InfoData/DcOutputShift
//     Drive/Inputs/In/nState1 <-> 1st TxPDO Mapping/Status Word
//     Drive/Inputs/In/nState2 <-> 1st TxPDO Mapping/Status Word @bit 8
//     Drive/Inputs/In/nState4 @bit 1 <-> WcState/InputToggle
//     Drive/Inputs/In/nState4 <-> WcState/WcState
//     Drive/Outputs/Out/nCtrl1 <-> 2nd RxPDO Mapping/Control Word
//     Drive/Outputs/Out/nCtrl2 <-> 2nd RxPDO Mapping/Control Word @bit 8
//     Drive/Outputs/Out/nDataOut1 <-> 2nd RxPDO Mapping/TargetPosition
//     Enc/Inputs/In/nDataIn1 <-> 1st TxPDO Mapping/ActualPosition
//     Enc/Inputs/In/nDataIn7 <-> 1st TxPDO Mapping/Velocity actual value
//     Enc/Inputs/In/nDcInputTime <-> InfoData/DcInputShift
//     Enc/Inputs/In/nState4 @bit 1 <-> WcState/InputToggle
//     Enc/Inputs/In/nState4 <-> WcState/WcState
//   NC-Task 1 SAF/Axes/Counter 31 <-> Device 4 (EtherCAT)/Drive PA13301 (ASDA-A2-E CoE Drive)
//     Drive/Inputs/In/nDataIn3[0] <-> 1st Transmit PDO Mapping/Torque actual value
//     Drive/Inputs/In/nDcOutputTime <-> InfoData/DcOutputShift
//     Drive/Inputs/In/nState1 <-> 1st Transmit PDO Mapping/Statusword
//     Drive/Inputs/In/nState2 <-> 1st Transmit PDO Mapping/Statusword @bit 8
//     Drive/Inputs/In/nState4 @bit 1 <-> WcState/InputToggle
//     Drive/Inputs/In/nState4 <-> WcState/WcState
//     Drive/Outputs/Out/nCtrl1 <-> 2nd Receive PDO Mapping/Controlword
//     Drive/Outputs/Out/nCtrl2 <-> 2nd Receive PDO Mapping/Controlword @bit 8
//     Drive/Outputs/Out/nDataOut1 <-> 2nd Receive PDO Mapping/Target position
//     Enc/Inputs/In/nDataIn1 <-> 1st Transmit PDO Mapping/Position actual value
//     Enc/Inputs/In/nDataIn7 <-> 1st Transmit PDO Mapping/Velocity actual value
//     Enc/Inputs/In/nDcInputTime <-> InfoData/DcInputShift
//     Enc/Inputs/In/nState4 @bit 1 <-> WcState/InputToggle
//     Enc/Inputs/In/nState4 <-> WcState/WcState
//   NC-Task 1 SAF/Axes/Counter 32 <-> Device 4 (EtherCAT)/Drive PA13401 (ASDA-A2-E CoE Drive)
//     Drive/Inputs/In/nDataIn3[0] <-> 1st Transmit PDO Mapping/Torque actual value
//     Drive/Inputs/In/nDcOutputTime <-> InfoData/DcOutputShift
//     Drive/Inputs/In/nState1 <-> 1st Transmit PDO Mapping/Statusword
//     Drive/Inputs/In/nState2 <-> 1st Transmit PDO Mapping/Statusword @bit 8
//     Drive/Inputs/In/nState4 @bit 1 <-> WcState/InputToggle
//     Drive/Inputs/In/nState4 <-> WcState/WcState
//     Drive/Outputs/Out/nCtrl1 <-> 2nd Receive PDO Mapping/Controlword
//     Drive/Outputs/Out/nCtrl2 <-> 2nd Receive PDO Mapping/Controlword @bit 8
//     Drive/Outputs/Out/nDataOut1 <-> 2nd Receive PDO Mapping/Target position
//     Enc/Inputs/In/nDataIn1 <-> 1st Transmit PDO Mapping/Position actual value
//     Enc/Inputs/In/nDataIn7 <-> 1st Transmit PDO Mapping/Velocity actual value
//     Enc/Inputs/In/nDcInputTime <-> InfoData/DcInputShift
//     Enc/Inputs/In/nState4 @bit 1 <-> WcState/InputToggle
//     Enc/Inputs/In/nState4 <-> WcState/WcState
//   NC-Task 1 SAF/Axes/Counter 33 <-> Device 4 (EtherCAT)/Drive PA13501 (ASDA-A2-E CoE Drive)
//     Drive/Inputs/In/nDataIn3[0] <-> 1st Transmit PDO Mapping/Torque actual value
//     Drive/Inputs/In/nDcOutputTime <-> InfoData/DcOutputShift
//     Drive/Inputs/In/nState1 <-> 1st Transmit PDO Mapping/Statusword
//     Drive/Inputs/In/nState2 <-> 1st Transmit PDO Mapping/Statusword @bit 8
//     Drive/Inputs/In/nState4 @bit 1 <-> WcState/InputToggle
//     Drive/Inputs/In/nState4 <-> WcState/WcState
//     Drive/Outputs/Out/nCtrl1 <-> 2nd Receive PDO Mapping/Controlword
//     Drive/Outputs/Out/nCtrl2 <-> 2nd Receive PDO Mapping/Controlword @bit 8
//     Drive/Outputs/Out/nDataOut1 <-> 2nd Receive PDO Mapping/Target position
//     Enc/Inputs/In/nDataIn1 <-> 1st Transmit PDO Mapping/Position actual value
//     Enc/Inputs/In/nDataIn7 <-> 1st Transmit PDO Mapping/Velocity actual value
//     Enc/Inputs/In/nDcInputTime <-> InfoData/DcInputShift
//     Enc/Inputs/In/nState4 @bit 1 <-> WcState/InputToggle
//     Enc/Inputs/In/nState4 <-> WcState/WcState
//   NC-Task 1 SAF/Axes/Counter 34 <-> Device 4 (EtherCAT)/Drive PA13601 (ASDA-A2-E CoE Drive)
//     Drive/Inputs/In/nDataIn3[0] <-> 1st TxPDO Mapping/ActualTorque
//     Drive/Inputs/In/nDcOutputTime <-> InfoData/DcOutputShift
//     Drive/Inputs/In/nState1 <-> 1st TxPDO Mapping/Status Word
//     Drive/Inputs/In/nState2 <-> 1st TxPDO Mapping/Status Word @bit 8
//     Drive/Inputs/In/nState4 @bit 1 <-> WcState/InputToggle
//     Drive/Inputs/In/nState4 <-> WcState/WcState
//     Drive/Outputs/Out/nCtrl1 <-> 2nd RxPDO Mapping/Control Word
//     Drive/Outputs/Out/nCtrl2 <-> 2nd RxPDO Mapping/Control Word @bit 8
//     Drive/Outputs/Out/nDataOut1 <-> 2nd RxPDO Mapping/TargetPosition
//     Enc/Inputs/In/nDataIn1 <-> 1st TxPDO Mapping/ActualPosition
//     Enc/Inputs/In/nDataIn7 <-> 1st TxPDO Mapping/Velocity actual value
//     Enc/Inputs/In/nDcInputTime <-> InfoData/DcInputShift
//     Enc/Inputs/In/nState4 @bit 1 <-> WcState/InputToggle
//     Enc/Inputs/In/nState4 <-> WcState/WcState
//   NC-Task 1 SAF/Axes/Counter 35 <-> Device 4 (EtherCAT)/Drive PA13701 (ASDA-A2-E CoE Drive)
//     Drive/Inputs/In/nDataIn3[0] <-> 1st TxPDO Mapping/ActualTorque
//     Drive/Inputs/In/nDcOutputTime <-> InfoData/DcOutputShift
//     Drive/Inputs/In/nState1 <-> 1st TxPDO Mapping/Status Word
//     Drive/Inputs/In/nState2 <-> 1st TxPDO Mapping/Status Word @bit 8
//     Drive/Inputs/In/nState4 @bit 1 <-> WcState/InputToggle
//     Drive/Inputs/In/nState4 <-> WcState/WcState
//     Drive/Outputs/Out/nCtrl1 <-> 2nd RxPDO Mapping/Control Word
//     Drive/Outputs/Out/nCtrl2 <-> 2nd RxPDO Mapping/Control Word @bit 8
//     Drive/Outputs/Out/nDataOut1 <-> 2nd RxPDO Mapping/TargetPosition
//     Enc/Inputs/In/nDataIn1 <-> 1st TxPDO Mapping/ActualPosition
//     Enc/Inputs/In/nDataIn7 <-> 1st TxPDO Mapping/Velocity actual value
//     Enc/Inputs/In/nDcInputTime <-> InfoData/DcInputShift
//     Enc/Inputs/In/nState4 @bit 1 <-> WcState/InputToggle
//     Enc/Inputs/In/nState4 <-> WcState/WcState
//   NC-Task 1 SAF/Axes/Counter 36 <-> Device 4 (EtherCAT)/Drive PA13801 (ASDA-A2-E CoE Drive)
//     Drive/Inputs/In/nDataIn3[0] <-> 1st TxPDO Mapping/ActualTorque
//     Drive/Inputs/In/nDcOutputTime <-> InfoData/DcOutputShift
//     Drive/Inputs/In/nState1 <-> 1st TxPDO Mapping/Status Word
//     Drive/Inputs/In/nState2 <-> 1st TxPDO Mapping/Status Word @bit 8
//     Drive/Inputs/In/nState4 @bit 1 <-> WcState/InputToggle
//     Drive/Inputs/In/nState4 <-> WcState/WcState
//     Drive/Outputs/Out/nCtrl1 <-> 2nd RxPDO Mapping/Control Word
//     Drive/Outputs/Out/nCtrl2 <-> 2nd RxPDO Mapping/Control Word @bit 8
//     Drive/Outputs/Out/nDataOut1 <-> 2nd RxPDO Mapping/TargetPosition
//     Enc/Inputs/In/nDataIn1 <-> 1st TxPDO Mapping/ActualPosition
//     Enc/Inputs/In/nDataIn7 <-> 1st TxPDO Mapping/Velocity actual value
//     Enc/Inputs/In/nDcInputTime <-> InfoData/DcInputShift
//     Enc/Inputs/In/nState4 @bit 1 <-> WcState/InputToggle
//     Enc/Inputs/In/nState4 <-> WcState/WcState
//   NC-Task 1 SAF/Axes/Counter 37 <-> Device 4 (EtherCAT)/Drive PA13901 (ASDA-A2-E CoE Drive)
//     Drive/Inputs/In/nDataIn3[0] <-> 1st TxPDO Mapping/ActualTorque
//     Drive/Inputs/In/nDcOutputTime <-> InfoData/DcOutputShift
//     Drive/Inputs/In/nState1 <-> 1st TxPDO Mapping/Status Word
//     Drive/Inputs/In/nState2 <-> 1st TxPDO Mapping/Status Word @bit 8
//     Drive/Inputs/In/nState4 @bit 1 <-> WcState/InputToggle
//     Drive/Inputs/In/nState4 <-> WcState/WcState
//     Drive/Outputs/Out/nCtrl1 <-> 2nd RxPDO Mapping/Control Word
//     Drive/Outputs/Out/nCtrl2 <-> 2nd RxPDO Mapping/Control Word @bit 8
//     Drive/Outputs/Out/nDataOut1 <-> 2nd RxPDO Mapping/TargetPosition
//     Enc/Inputs/In/nDataIn1 <-> 1st TxPDO Mapping/ActualPosition
//     Enc/Inputs/In/nDataIn7 <-> 1st TxPDO Mapping/Velocity actual value
//     Enc/Inputs/In/nDcInputTime <-> InfoData/DcInputShift
//     Enc/Inputs/In/nState4 @bit 1 <-> WcState/InputToggle
//     Enc/Inputs/In/nState4 <-> WcState/WcState
//   NC-Task 1 SAF/Axes/Counter 38 <-> Device 4 (EtherCAT)/Drive PA14001 (ASDA-A2-E CoE Drive)
//     Drive/Inputs/In/nDataIn3[0] <-> 1st TxPDO Mapping/ActualTorque
//     Drive/Inputs/In/nDcOutputTime <-> InfoData/DcOutputShift
//     Drive/Inputs/In/nState1 <-> 1st TxPDO Mapping/Status Word
//     Drive/Inputs/In/nState2 <-> 1st TxPDO Mapping/Status Word @bit 8
//     Drive/Inputs/In/nState4 @bit 1 <-> WcState/InputToggle
//     Drive/Inputs/In/nState4 <-> WcState/WcState
//     Drive/Outputs/Out/nCtrl1 <-> 2nd RxPDO Mapping/Control Word
//     Drive/Outputs/Out/nCtrl2 <-> 2nd RxPDO Mapping/Control Word @bit 8
//     Drive/Outputs/Out/nDataOut1 <-> 2nd RxPDO Mapping/TargetPosition
//     Enc/Inputs/In/nDataIn1 <-> 1st TxPDO Mapping/ActualPosition
//     Enc/Inputs/In/nDataIn7 <-> 1st TxPDO Mapping/Velocity actual value
//     Enc/Inputs/In/nDcInputTime <-> InfoData/DcInputShift
//     Enc/Inputs/In/nState4 @bit 1 <-> WcState/InputToggle
//     Enc/Inputs/In/nState4 <-> WcState/WcState
//   NC-Task 1 SAF/Axes/Counter 39 <-> Device 4 (EtherCAT)/Drive PA14101 (ASDA-A2-E CoE Drive)
//     Drive/Inputs/In/nDataIn3[0] <-> 1st TxPDO Mapping/ActualTorque
//     Drive/Inputs/In/nDcOutputTime <-> InfoData/DcOutputShift
//     Drive/Inputs/In/nState1 <-> 1st TxPDO Mapping/Status Word
//     Drive/Inputs/In/nState2 <-> 1st TxPDO Mapping/Status Word @bit 8
//     Drive/Inputs/In/nState4 @bit 1 <-> WcState/InputToggle
//     Drive/Inputs/In/nState4 <-> WcState/WcState
//     Drive/Outputs/Out/nCtrl1 <-> 2nd RxPDO Mapping/Control Word
//     Drive/Outputs/Out/nCtrl2 <-> 2nd RxPDO Mapping/Control Word @bit 8
//     Drive/Outputs/Out/nDataOut1 <-> 2nd RxPDO Mapping/TargetPosition
//     Enc/Inputs/In/nDataIn1 <-> 1st TxPDO Mapping/ActualPosition
//     Enc/Inputs/In/nDataIn7 <-> 1st TxPDO Mapping/Velocity actual value
//     Enc/Inputs/In/nDcInputTime <-> InfoData/DcInputShift
//     Enc/Inputs/In/nState4 @bit 1 <-> WcState/InputToggle
//     Enc/Inputs/In/nState4 <-> WcState/WcState
//   NC-Task 1 SAF/Axes/Counter 4 <-> Device 4 (EtherCAT)/Drive PA10401 (ASDA-A2-E CoE Drive)
//     Drive/Inputs/In/nDataIn3[0] <-> 1st TxPDO Mapping/ActualTorque
//     Drive/Inputs/In/nDcOutputTime <-> InfoData/DcOutputShift
//     Drive/Inputs/In/nState1 <-> 1st TxPDO Mapping/Status Word
//     Drive/Inputs/In/nState2 <-> 1st TxPDO Mapping/Status Word @bit 8
//     Drive/Inputs/In/nState4 @bit 1 <-> WcState/InputToggle
//     Drive/Inputs/In/nState4 <-> WcState/WcState
//     Drive/Outputs/Out/nCtrl1 <-> 2nd RxPDO Mapping/Control Word
//     Drive/Outputs/Out/nCtrl2 <-> 2nd RxPDO Mapping/Control Word @bit 8
//     Drive/Outputs/Out/nDataOut1 <-> 2nd RxPDO Mapping/TargetPosition
//     Enc/Inputs/In/nDataIn1 <-> 1st TxPDO Mapping/ActualPosition
//     Enc/Inputs/In/nDataIn7 <-> 1st TxPDO Mapping/Velocity actual value
//     Enc/Inputs/In/nDcInputTime <-> InfoData/DcInputShift
//     Enc/Inputs/In/nState4 @bit 1 <-> WcState/InputToggle
//     Enc/Inputs/In/nState4 <-> WcState/WcState
//   NC-Task 1 SAF/Axes/Counter 40 <-> Device 4 (EtherCAT)/Drive PA14201 (ASDA-A2-E CoE Drive)
//     Drive/Inputs/In/nDataIn3[0] <-> 1st TxPDO Mapping/ActualTorque
//     Drive/Inputs/In/nDcOutputTime <-> InfoData/DcOutputShift
//     Drive/Inputs/In/nState1 <-> 1st TxPDO Mapping/Status Word
//     Drive/Inputs/In/nState2 <-> 1st TxPDO Mapping/Status Word @bit 8
//     Drive/Inputs/In/nState4 @bit 1 <-> WcState/InputToggle
//     Drive/Inputs/In/nState4 <-> WcState/WcState
//     Drive/Outputs/Out/nCtrl1 <-> 2nd RxPDO Mapping/Control Word
//     Drive/Outputs/Out/nCtrl2 <-> 2nd RxPDO Mapping/Control Word @bit 8
//     Drive/Outputs/Out/nDataOut1 <-> 2nd RxPDO Mapping/TargetPosition
//     Enc/Inputs/In/nDataIn1 <-> 1st TxPDO Mapping/ActualPosition
//     Enc/Inputs/In/nDataIn7 <-> 1st TxPDO Mapping/Velocity actual value
//     Enc/Inputs/In/nDcInputTime <-> InfoData/DcInputShift
//     Enc/Inputs/In/nState4 @bit 1 <-> WcState/InputToggle
//     Enc/Inputs/In/nState4 <-> WcState/WcState
//   NC-Task 1 SAF/Axes/Counter 5 <-> Device 4 (EtherCAT)/Drive PA10501 (ASDA-A2-E CoE Drive)
//     Drive/Inputs/In/nDataIn3[0] <-> 1st TxPDO Mapping/ActualTorque
//     Drive/Inputs/In/nDcOutputTime <-> InfoData/DcOutputShift
//     Drive/Inputs/In/nState1 <-> 1st TxPDO Mapping/Status Word
//     Drive/Inputs/In/nState2 <-> 1st TxPDO Mapping/Status Word @bit 8
//     Drive/Inputs/In/nState4 @bit 1 <-> WcState/InputToggle
//     Drive/Inputs/In/nState4 <-> WcState/WcState
//     Drive/Outputs/Out/nCtrl1 <-> 2nd RxPDO Mapping/Control Word
//     Drive/Outputs/Out/nCtrl2 <-> 2nd RxPDO Mapping/Control Word @bit 8
//     Drive/Outputs/Out/nDataOut1 <-> 2nd RxPDO Mapping/TargetPosition
//     Enc/Inputs/In/nDataIn1 <-> 1st TxPDO Mapping/ActualPosition
//     Enc/Inputs/In/nDataIn7 <-> 1st TxPDO Mapping/Velocity actual value
//     Enc/Inputs/In/nDcInputTime <-> InfoData/DcInputShift
//     Enc/Inputs/In/nState4 @bit 1 <-> WcState/InputToggle
//     Enc/Inputs/In/nState4 <-> WcState/WcState
//   NC-Task 1 SAF/Axes/Counter 6 <-> Device 4 (EtherCAT)/Drive PA10601 (ASDA-A2-E CoE Drive)
//     Drive/Inputs/In/nDataIn3[0] <-> 1st TxPDO Mapping/ActualTorque
//     Drive/Inputs/In/nDcOutputTime <-> InfoData/DcOutputShift
//     Drive/Inputs/In/nState1 <-> 1st TxPDO Mapping/Status Word
//     Drive/Inputs/In/nState2 <-> 1st TxPDO Mapping/Status Word @bit 8
//     Drive/Inputs/In/nState4 @bit 1 <-> WcState/InputToggle
//     Drive/Inputs/In/nState4 <-> WcState/WcState
//     Drive/Outputs/Out/nCtrl1 <-> 2nd RxPDO Mapping/Control Word
//     Drive/Outputs/Out/nCtrl2 <-> 2nd RxPDO Mapping/Control Word @bit 8
//     Drive/Outputs/Out/nDataOut1 <-> 2nd RxPDO Mapping/TargetPosition
//     Enc/Inputs/In/nDataIn1 <-> 1st TxPDO Mapping/ActualPosition
//     Enc/Inputs/In/nDataIn7 <-> 1st TxPDO Mapping/Velocity actual value
//     Enc/Inputs/In/nDcInputTime <-> InfoData/DcInputShift
//     Enc/Inputs/In/nState4 @bit 1 <-> WcState/InputToggle
//     Enc/Inputs/In/nState4 <-> WcState/WcState
//   NC-Task 1 SAF/Axes/Counter 7 <-> Device 4 (EtherCAT)/Drive PA10701 (ASDA-A2-E CoE Drive)
//     Drive/Inputs/In/nDataIn3[0] <-> 1st TxPDO Mapping/ActualTorque
//     Drive/Inputs/In/nDcOutputTime <-> InfoData/DcOutputShift
//     Drive/Inputs/In/nState1 <-> 1st TxPDO Mapping/Status Word
//     Drive/Inputs/In/nState2 <-> 1st TxPDO Mapping/Status Word @bit 8
//     Drive/Inputs/In/nState4 @bit 1 <-> WcState/InputToggle
//     Drive/Inputs/In/nState4 <-> WcState/WcState
//     Drive/Outputs/Out/nCtrl1 <-> 2nd RxPDO Mapping/Control Word
//     Drive/Outputs/Out/nCtrl2 <-> 2nd RxPDO Mapping/Control Word @bit 8
//     Drive/Outputs/Out/nDataOut1 <-> 2nd RxPDO Mapping/TargetPosition
//     Enc/Inputs/In/nDataIn1 <-> 1st TxPDO Mapping/ActualPosition
//     Enc/Inputs/In/nDataIn7 <-> 1st TxPDO Mapping/Velocity actual value
//     Enc/Inputs/In/nDcInputTime <-> InfoData/DcInputShift
//     Enc/Inputs/In/nState4 @bit 1 <-> WcState/InputToggle
//     Enc/Inputs/In/nState4 <-> WcState/WcState
//   NC-Task 1 SAF/Axes/Counter 8 <-> Device 4 (EtherCAT)/Drive PA10801 (ASDA-A2-E CoE Drive)
//     Drive/Inputs/In/nDataIn3[0] <-> 1st TxPDO Mapping/ActualTorque
//     Drive/Inputs/In/nDcOutputTime <-> InfoData/DcOutputShift
//     Drive/Inputs/In/nState1 <-> 1st TxPDO Mapping/Status Word
//     Drive/Inputs/In/nState2 <-> 1st TxPDO Mapping/Status Word @bit 8
//     Drive/Inputs/In/nState4 @bit 1 <-> WcState/InputToggle
//     Drive/Inputs/In/nState4 <-> WcState/WcState
//     Drive/Outputs/Out/nCtrl1 <-> 2nd RxPDO Mapping/Control Word
//     Drive/Outputs/Out/nCtrl2 <-> 2nd RxPDO Mapping/Control Word @bit 8
//     Drive/Outputs/Out/nDataOut1 <-> 2nd RxPDO Mapping/TargetPosition
//     Enc/Inputs/In/nDataIn1 <-> 1st TxPDO Mapping/ActualPosition
//     Enc/Inputs/In/nDataIn7 <-> 1st TxPDO Mapping/Velocity actual value
//     Enc/Inputs/In/nDcInputTime <-> InfoData/DcInputShift
//     Enc/Inputs/In/nState4 @bit 1 <-> WcState/InputToggle
//     Enc/Inputs/In/nState4 <-> WcState/WcState
//   NC-Task 1 SAF/Axes/Counter 9 <-> Device 4 (EtherCAT)/Drive PA10901 (ASDA-A2-E CoE Drive)
//     Drive/Inputs/In/nDataIn3[0] <-> 1st TxPDO Mapping/ActualTorque
//     Drive/Inputs/In/nDcOutputTime <-> InfoData/DcOutputShift
//     Drive/Inputs/In/nState1 <-> 1st TxPDO Mapping/Status Word
//     Drive/Inputs/In/nState2 <-> 1st TxPDO Mapping/Status Word @bit 8
//     Drive/Inputs/In/nState4 @bit 1 <-> WcState/InputToggle
//     Drive/Inputs/In/nState4 <-> WcState/WcState
//     Drive/Outputs/Out/nCtrl1 <-> 2nd RxPDO Mapping/Control Word
//     Drive/Outputs/Out/nCtrl2 <-> 2nd RxPDO Mapping/Control Word @bit 8
//     Drive/Outputs/Out/nDataOut1 <-> 2nd RxPDO Mapping/TargetPosition
//     Enc/Inputs/In/nDataIn1 <-> 1st TxPDO Mapping/ActualPosition
//     Enc/Inputs/In/nDataIn7 <-> 1st TxPDO Mapping/Velocity actual value
//     Enc/Inputs/In/nDcInputTime <-> InfoData/DcInputShift
//     Enc/Inputs/In/nState4 @bit 1 <-> WcState/InputToggle
//     Enc/Inputs/In/nState4 <-> WcState/WcState
//   NC-Task 1 SAF/Axes/Puller <-> Device 1 (EtherCAT)/Term 1 (EK1200)/Term 17 (EK1122)/Drive PA14701 (ASDA-A2-E CoE Drive)
//     Drive/Inputs/In/nDataIn3[0] <-> 1st Transmit PDO Mapping/Torque actual value
//     Drive/Inputs/In/nDcOutputTime <-> InfoData/DcOutputShift
//     Drive/Inputs/In/nState1 <-> 1st Transmit PDO Mapping/Statusword
//     Drive/Inputs/In/nState2 <-> 1st Transmit PDO Mapping/Statusword @bit 8
//     Drive/Inputs/In/nState4 @bit 1 <-> WcState/InputToggle
//     Drive/Inputs/In/nState4 <-> WcState/WcState
//     Drive/Outputs/Out/nCtrl1 <-> 2nd Receive PDO Mapping/Controlword
//     Drive/Outputs/Out/nCtrl2 <-> 2nd Receive PDO Mapping/Controlword @bit 8
//     Drive/Outputs/Out/nDataOut1 <-> 2nd Receive PDO Mapping/Target position
//     Enc/Inputs/In/nDataIn1 <-> 1st Transmit PDO Mapping/Position actual value
//     Enc/Inputs/In/nDataIn7 <-> 1st Transmit PDO Mapping/Velocity actual value
//     Enc/Inputs/In/nDcInputTime <-> InfoData/DcInputShift
//     Enc/Inputs/In/nState4 @bit 1 <-> WcState/InputToggle
//     Enc/Inputs/In/nState4 <-> WcState/WcState
//   NC-Task 1 SAF/Axes/eAxis1 <-> Device 1 (EtherCAT)/Term 1 (EK1200)/Term 16 (EL5101)
//     Enc/Inputs/In/nDataIn1[0] <-> ENC Status compact/Counter value
//     Enc/Inputs/In/nDataIn2[0] <-> ENC Status compact/Latch value
//     Enc/Inputs/In/nState1 @bit 4 <-> ENC Status compact/Status/Counter overflow
//     Enc/Inputs/In/nState1 @bit 3 <-> ENC Status compact/Status/Counter underflow
//     Enc/Inputs/In/nState1 @bit 7 <-> ENC Status compact/Status/Extrapolation stall
//     Enc/Inputs/In/nState1 <-> ENC Status compact/Status/Latch C valid
//     Enc/Inputs/In/nState1 @bit 1 <-> ENC Status compact/Status/Latch extern valid
//     Enc/Inputs/In/nState1 @bit 6 <-> ENC Status compact/Status/Open circuit
//     Enc/Inputs/In/nState1 @bit 2 <-> ENC Status compact/Status/Set counter done
//     Enc/Inputs/In/nState1 @bit 5 <-> ENC Status compact/Status/Status of input status
//     Enc/Inputs/In/nState2 @bit 4 <-> ENC Status compact/Status/Status of extern latch
//     Enc/Inputs/In/nState2 <-> ENC Status compact/Status/Status of input A
//     Enc/Inputs/In/nState2 @bit 1 <-> ENC Status compact/Status/Status of input B
//     Enc/Inputs/In/nState2 @bit 2 <-> ENC Status compact/Status/Status of input C
//     Enc/Inputs/In/nState2 @bit 3 <-> ENC Status compact/Status/Status of input gate
//     Enc/Inputs/In/nState2 @bit 5 <-> ENC Status compact/Status/Sync error
//     Enc/Inputs/In/nState2 @bit 6 <-> ENC Status compact/Status/TxPDO State
//     Enc/Inputs/In/nState2 @bit 7 <-> ENC Status compact/Status/TxPDO Toggle
//     Enc/Inputs/In/nState4 @bit 1 <-> WcState/InputToggle
//     Enc/Inputs/In/nState4 <-> WcState/WcState
//     Enc/Outputs/Out/nCtrl1 <-> ENC Control compact/Control/Enable latch C
//     Enc/Outputs/Out/nCtrl1 @bit 3 <-> ENC Control compact/Control/Enable latch extern on negative edge
//     Enc/Outputs/Out/nCtrl1 @bit 1 <-> ENC Control compact/Control/Enable latch extern on positive edge
//     Enc/Outputs/Out/nCtrl1 @bit 2 <-> ENC Control compact/Control/Set counter
//     Enc/Outputs/Out/nDataOut1[0] <-> ENC Control compact/Set counter value
//   PLC1/PLC1 Instance <-> Device 1 (EtherCAT)
//     CommunicationTask Inputs/EtherCatStates.Device1_nEcMasterDeviceId <-> InfoData/DevId
//     CommunicationTask Inputs/EtherCatStates.Device1_netID <-> InfoData/AmsNetId
//   PLC1/PLC1 Instance <-> Device 1 (EtherCAT)/Drive PA14901 (ASDA-A2-E CoE Drive)
//     PlcTask1 Inputs/ControllerTags.arErrorCodeDrive[48] <-> 1st TxPDO Mapping/Error code
//   PLC1/PLC1 Instance <-> Device 1 (EtherCAT)/Term 1 (EK1200)/Term 10 (EL2008)
//     IOTask Outputs/ControllerTags.EL2008[32,{1..8}] <-> Channel {1..8}/Output  (8 links)
//   PLC1/PLC1 Instance <-> Device 1 (EtherCAT)/Term 1 (EK1200)/Term 12 (EL3312)
//     PlcTask1 Inputs/ControllerTags.EL3312[1,1]/Status <-> TC Inputs Channel 1/Status
//     PlcTask1 Inputs/ControllerTags.EL3312[1,2]/Status <-> TC Inputs Channel 2/Status
//     PlcTask1 Inputs/ControllerTags.EL3312[1,1]/Value <-> TC Inputs Channel 1/Value
//     PlcTask1 Inputs/ControllerTags.EL3312[1,2]/Value <-> TC Inputs Channel 2/Value
//   PLC1/PLC1 Instance <-> Device 1 (EtherCAT)/Term 1 (EK1200)/Term 13 (EL3312)
//     PlcTask1 Inputs/ControllerTags.EL3312[2,1]/Status <-> TC Inputs Channel 1/Status
//     PlcTask1 Inputs/ControllerTags.EL3312[2,2]/Status <-> TC Inputs Channel 2/Status
//     PlcTask1 Inputs/ControllerTags.EL3312[2,1]/Value <-> TC Inputs Channel 1/Value
//     PlcTask1 Inputs/ControllerTags.EL3312[2,2]/Value <-> TC Inputs Channel 2/Value
//   PLC1/PLC1 Instance <-> Device 1 (EtherCAT)/Term 1 (EK1200)/Term 14 (EL3312)
//     PlcTask1 Inputs/ControllerTags.EL3312[3,1]/Status <-> TC Inputs Channel 1/Status
//     PlcTask1 Inputs/ControllerTags.EL3312[3,2]/Status <-> TC Inputs Channel 2/Status
//     PlcTask1 Inputs/ControllerTags.EL3312[3,1]/Value <-> TC Inputs Channel 1/Value
//     PlcTask1 Inputs/ControllerTags.EL3312[3,2]/Value <-> TC Inputs Channel 2/Value
//   PLC1/PLC1 Instance <-> Device 1 (EtherCAT)/Term 1 (EK1200)/Term 15 (EL3312)
//     PlcTask1 Inputs/ControllerTags.EL3312[4,1]/Status <-> TC Inputs Channel 1/Status
//     PlcTask1 Inputs/ControllerTags.EL3312[4,2]/Status <-> TC Inputs Channel 2/Status
//     PlcTask1 Inputs/ControllerTags.EL3312[4,1]/Value <-> TC Inputs Channel 1/Value
//     PlcTask1 Inputs/ControllerTags.EL3312[4,2]/Value <-> TC Inputs Channel 2/Value
//   PLC1/PLC1 Instance <-> Device 1 (EtherCAT)/Term 1 (EK1200)/Term 17 (EK1122)/CPX_1 VI45001 (CPX-AP-I-EC-M12)
//     IOTask Inputs/ControllerTags.CPX8_1[1,1] <-> Module 2 (CPX-AP-I-8DI-M8-3P)/Inputs/Input 0
//     IOTask Inputs/ControllerTags.CPX8_1[1,2] <-> Module 2 (CPX-AP-I-8DI-M8-3P)/Inputs/Input 1
//     IOTask Inputs/ControllerTags.CPX8_1[1,3] <-> Module 2 (CPX-AP-I-8DI-M8-3P)/Inputs/Input 2
//     IOTask Inputs/ControllerTags.CPX8_1[1,4] <-> Module 2 (CPX-AP-I-8DI-M8-3P)/Inputs/Input 3
//     IOTask Inputs/ControllerTags.CPX8_1[1,5] <-> Module 2 (CPX-AP-I-8DI-M8-3P)/Inputs/Input 4
//     IOTask Inputs/ControllerTags.CPX8_1[1,6] <-> Module 2 (CPX-AP-I-8DI-M8-3P)/Inputs/Input 5
//     IOTask Inputs/ControllerTags.CPX8_1[1,7] <-> Module 2 (CPX-AP-I-8DI-M8-3P)/Inputs/Input 6
//     IOTask Inputs/ControllerTags.CPX8_1[1,8] <-> Module 2 (CPX-AP-I-8DI-M8-3P)/Inputs/Input 7
//     IOTask Inputs/ControllerTags.CPX8_1[2,1] <-> Module 3 (CPX-AP-I-8DI-M8-3P)/Inputs/Input 0
//     IOTask Inputs/ControllerTags.CPX8_1[2,2] <-> Module 3 (CPX-AP-I-8DI-M8-3P)/Inputs/Input 1
//     IOTask Inputs/ControllerTags.CPX8_1[2,3] <-> Module 3 (CPX-AP-I-8DI-M8-3P)/Inputs/Input 2
//     IOTask Inputs/ControllerTags.CPX8_1[2,4] <-> Module 3 (CPX-AP-I-8DI-M8-3P)/Inputs/Input 3
//     IOTask Inputs/ControllerTags.CPX8_1[2,5] <-> Module 3 (CPX-AP-I-8DI-M8-3P)/Inputs/Input 4
//     IOTask Inputs/ControllerTags.CPX8_1[2,6] <-> Module 3 (CPX-AP-I-8DI-M8-3P)/Inputs/Input 5
//     IOTask Inputs/ControllerTags.CPX8_1[2,7] <-> Module 3 (CPX-AP-I-8DI-M8-3P)/Inputs/Input 6
//     IOTask Inputs/ControllerTags.CPX8_1[2,8] <-> Module 3 (CPX-AP-I-8DI-M8-3P)/Inputs/Input 7
//     IOTask Inputs/ControllerTags.CPX8_1[3,1] <-> Module 4 (CPX-AP-I-8DI-M8-3P)/Inputs/Input 0
//     IOTask Inputs/ControllerTags.CPX8_1[3,2] <-> Module 4 (CPX-AP-I-8DI-M8-3P)/Inputs/Input 1
//     IOTask Inputs/ControllerTags.CPX8_1[3,3] <-> Module 4 (CPX-AP-I-8DI-M8-3P)/Inputs/Input 2
//     IOTask Inputs/ControllerTags.CPX8_1[3,4] <-> Module 4 (CPX-AP-I-8DI-M8-3P)/Inputs/Input 3
//     IOTask Inputs/ControllerTags.CPX8_1[3,5] <-> Module 4 (CPX-AP-I-8DI-M8-3P)/Inputs/Input 4
//     IOTask Inputs/ControllerTags.CPX8_1[3,6] <-> Module 4 (CPX-AP-I-8DI-M8-3P)/Inputs/Input 5
//     IOTask Inputs/ControllerTags.CPX8_1[3,7] <-> Module 4 (CPX-AP-I-8DI-M8-3P)/Inputs/Input 6
//     IOTask Inputs/ControllerTags.CPX8_1[3,8] <-> Module 4 (CPX-AP-I-8DI-M8-3P)/Inputs/Input 7
//     IOTask Inputs/ControllerTags.CPX8_1[4,1] <-> Module 5 (CPX-AP-I-8DI-M8-3P)/Inputs/Input 0
//     IOTask Inputs/ControllerTags.CPX8_1[4,2] <-> Module 5 (CPX-AP-I-8DI-M8-3P)/Inputs/Input 1
//     IOTask Inputs/ControllerTags.CPX8_1[4,3] <-> Module 5 (CPX-AP-I-8DI-M8-3P)/Inputs/Input 2
//     IOTask Inputs/ControllerTags.CPX8_1[4,4] <-> Module 5 (CPX-AP-I-8DI-M8-3P)/Inputs/Input 3
//     IOTask Inputs/ControllerTags.CPX8_1[4,5] <-> Module 5 (CPX-AP-I-8DI-M8-3P)/Inputs/Input 4
//     IOTask Inputs/ControllerTags.CPX8_1[4,6] <-> Module 5 (CPX-AP-I-8DI-M8-3P)/Inputs/Input 5
//     IOTask Inputs/ControllerTags.CPX8_1[4,7] <-> Module 5 (CPX-AP-I-8DI-M8-3P)/Inputs/Input 6
//     IOTask Inputs/ControllerTags.CPX8_1[4,8] <-> Module 5 (CPX-AP-I-8DI-M8-3P)/Inputs/Input 7
//     IOTask Inputs/ControllerTags.CPX8_1[5,1] <-> Module 6 (CPX-AP-I-8DI-M8-3P)/Inputs/Input 0
//     IOTask Inputs/ControllerTags.CPX8_1[5,2] <-> Module 6 (CPX-AP-I-8DI-M8-3P)/Inputs/Input 1
//     IOTask Inputs/ControllerTags.CPX8_1[5,3] <-> Module 6 (CPX-AP-I-8DI-M8-3P)/Inputs/Input 2
//     IOTask Inputs/ControllerTags.CPX8_1[5,4] <-> Module 6 (CPX-AP-I-8DI-M8-3P)/Inputs/Input 3
//     IOTask Inputs/ControllerTags.CPX8_1[5,5] <-> Module 6 (CPX-AP-I-8DI-M8-3P)/Inputs/Input 4
//     IOTask Inputs/ControllerTags.CPX8_1[5,6] <-> Module 6 (CPX-AP-I-8DI-M8-3P)/Inputs/Input 5
//     IOTask Inputs/ControllerTags.CPX8_1[5,7] <-> Module 6 (CPX-AP-I-8DI-M8-3P)/Inputs/Input 6
//     IOTask Inputs/ControllerTags.CPX8_1[5,8] <-> Module 6 (CPX-AP-I-8DI-M8-3P)/Inputs/Input 7
//     IOTask Inputs/ControllerTags.CPX8_1[6,1] <-> Module 7 (CPX-AP-I-8DI-M8-3P)/Inputs/Input 0
//     IOTask Inputs/ControllerTags.CPX8_1[6,2] <-> Module 7 (CPX-AP-I-8DI-M8-3P)/Inputs/Input 1
//     IOTask Inputs/ControllerTags.CPX8_1[6,3] <-> Module 7 (CPX-AP-I-8DI-M8-3P)/Inputs/Input 2
//     IOTask Inputs/ControllerTags.CPX8_1[6,4] <-> Module 7 (CPX-AP-I-8DI-M8-3P)/Inputs/Input 3
//     IOTask Inputs/ControllerTags.CPX8_1[6,5] <-> Module 7 (CPX-AP-I-8DI-M8-3P)/Inputs/Input 4
